   // UNICODE_TO_GBK[29826] := 16#8574;
   // UNICODE_TO_GBK[29827] := 16#D4CC;
   // UNICODE_TO_GBK[29828] := 16#8575;
   // UNICODE_TO_GBK[29829] := 16#CA98;
   // UNICODE_TO_GBK[29830] := 16#8576;
   // UNICODE_TO_GBK[29831] := 16#CA99;
   // UNICODE_TO_GBK[29832] := 16#8577;
   // UNICODE_TO_GBK[29833] := 16#CA9A;
   // UNICODE_TO_GBK[29834] := 16#8578;
   // UNICODE_TO_GBK[29835] := 16#CA9B;
   // UNICODE_TO_GBK[29836] := 16#8579;
   // UNICODE_TO_GBK[29837] := 16#DEB3;
   // UNICODE_TO_GBK[29838] := 16#857A;
   // UNICODE_TO_GBK[29839] := 16#DEAA;
   // UNICODE_TO_GBK[29840] := 16#857B;
   // UNICODE_TO_GBK[29841] := 16#DEAE;
   // UNICODE_TO_GBK[29842] := 16#857C;
   // UNICODE_TO_GBK[29843] := 16#CA9C;
   // UNICODE_TO_GBK[29844] := 16#857D;
   // UNICODE_TO_GBK[29845] := 16#CA9D;
   // UNICODE_TO_GBK[29846] := 16#857E;
   // UNICODE_TO_GBK[29847] := 16#C0D9;
   // UNICODE_TO_GBK[29848] := 16#857F;
   // UNICODE_TO_GBK[29849] := 16#CA9E;
   // UNICODE_TO_GBK[29850] := 16#8580;
   // UNICODE_TO_GBK[29851] := 16#CA9F;
   // UNICODE_TO_GBK[29852] := 16#8581;
   // UNICODE_TO_GBK[29853] := 16#CAA0;
   // UNICODE_TO_GBK[29854] := 16#8582;
   // UNICODE_TO_GBK[29855] := 16#CB40;
   // UNICODE_TO_GBK[29856] := 16#8583;
   // UNICODE_TO_GBK[29857] := 16#CB41;
   // UNICODE_TO_GBK[29858] := 16#8584;
   // UNICODE_TO_GBK[29859] := 16#B1A1;
   // UNICODE_TO_GBK[29860] := 16#8585;
   // UNICODE_TO_GBK[29861] := 16#DEB6;
   // UNICODE_TO_GBK[29862] := 16#8586;
   // UNICODE_TO_GBK[29863] := 16#CB42;
   // UNICODE_TO_GBK[29864] := 16#8587;
   // UNICODE_TO_GBK[29865] := 16#DEB1;
   // UNICODE_TO_GBK[29866] := 16#8588;
   // UNICODE_TO_GBK[29867] := 16#CB43;
   // UNICODE_TO_GBK[29868] := 16#8589;
   // UNICODE_TO_GBK[29869] := 16#CB44;
   // UNICODE_TO_GBK[29870] := 16#858A;
   // UNICODE_TO_GBK[29871] := 16#CB45;
   // UNICODE_TO_GBK[29872] := 16#858B;
   // UNICODE_TO_GBK[29873] := 16#CB46;
   // UNICODE_TO_GBK[29874] := 16#858C;
   // UNICODE_TO_GBK[29875] := 16#CB47;
   // UNICODE_TO_GBK[29876] := 16#858D;
   // UNICODE_TO_GBK[29877] := 16#CB48;
   // UNICODE_TO_GBK[29878] := 16#858E;
   // UNICODE_TO_GBK[29879] := 16#CB49;
   // UNICODE_TO_GBK[29880] := 16#858F;
   // UNICODE_TO_GBK[29881] := 16#DEB2;
   // UNICODE_TO_GBK[29882] := 16#8590;
   // UNICODE_TO_GBK[29883] := 16#CB4A;
   // UNICODE_TO_GBK[29884] := 16#8591;
   // UNICODE_TO_GBK[29885] := 16#CB4B;
   // UNICODE_TO_GBK[29886] := 16#8592;
   // UNICODE_TO_GBK[29887] := 16#CB4C;
   // UNICODE_TO_GBK[29888] := 16#8593;
   // UNICODE_TO_GBK[29889] := 16#CB4D;
   // UNICODE_TO_GBK[29890] := 16#8594;
   // UNICODE_TO_GBK[29891] := 16#CB4E;
   // UNICODE_TO_GBK[29892] := 16#8595;
   // UNICODE_TO_GBK[29893] := 16#CB4F;
   // UNICODE_TO_GBK[29894] := 16#8596;
   // UNICODE_TO_GBK[29895] := 16#CB50;
   // UNICODE_TO_GBK[29896] := 16#8597;
   // UNICODE_TO_GBK[29897] := 16#CB51;
   // UNICODE_TO_GBK[29898] := 16#8598;
   // UNICODE_TO_GBK[29899] := 16#CB52;
   // UNICODE_TO_GBK[29900] := 16#8599;
   // UNICODE_TO_GBK[29901] := 16#CB53;
   // UNICODE_TO_GBK[29902] := 16#859A;
   // UNICODE_TO_GBK[29903] := 16#CB54;
   // UNICODE_TO_GBK[29904] := 16#859B;
   // UNICODE_TO_GBK[29905] := 16#D1A6;
   // UNICODE_TO_GBK[29906] := 16#859C;
   // UNICODE_TO_GBK[29907] := 16#DEB5;
   // UNICODE_TO_GBK[29908] := 16#859D;
   // UNICODE_TO_GBK[29909] := 16#CB55;
   // UNICODE_TO_GBK[29910] := 16#859E;
   // UNICODE_TO_GBK[29911] := 16#CB56;
   // UNICODE_TO_GBK[29912] := 16#859F;
   // UNICODE_TO_GBK[29913] := 16#CB57;
   // UNICODE_TO_GBK[29914] := 16#85A0;
   // UNICODE_TO_GBK[29915] := 16#CB58;
   // UNICODE_TO_GBK[29916] := 16#85A1;
   // UNICODE_TO_GBK[29917] := 16#CB59;
   // UNICODE_TO_GBK[29918] := 16#85A2;
   // UNICODE_TO_GBK[29919] := 16#CB5A;
   // UNICODE_TO_GBK[29920] := 16#85A3;
   // UNICODE_TO_GBK[29921] := 16#CB5B;
   // UNICODE_TO_GBK[29922] := 16#85A4;
   // UNICODE_TO_GBK[29923] := 16#DEAF;
   // UNICODE_TO_GBK[29924] := 16#85A5;
   // UNICODE_TO_GBK[29925] := 16#CB5C;
   // UNICODE_TO_GBK[29926] := 16#85A6;
   // UNICODE_TO_GBK[29927] := 16#CB5D;
   // UNICODE_TO_GBK[29928] := 16#85A7;
   // UNICODE_TO_GBK[29929] := 16#CB5E;
   // UNICODE_TO_GBK[29930] := 16#85A8;
   // UNICODE_TO_GBK[29931] := 16#DEB0;
   // UNICODE_TO_GBK[29932] := 16#85A9;
   // UNICODE_TO_GBK[29933] := 16#CB5F;
   // UNICODE_TO_GBK[29934] := 16#85AA;
   // UNICODE_TO_GBK[29935] := 16#D0BD;
   // UNICODE_TO_GBK[29936] := 16#85AB;
   // UNICODE_TO_GBK[29937] := 16#CB60;
   // UNICODE_TO_GBK[29938] := 16#85AC;
   // UNICODE_TO_GBK[29939] := 16#CB61;
   // UNICODE_TO_GBK[29940] := 16#85AD;
   // UNICODE_TO_GBK[29941] := 16#CB62;
   // UNICODE_TO_GBK[29942] := 16#85AE;
   // UNICODE_TO_GBK[29943] := 16#DEB4;
   // UNICODE_TO_GBK[29944] := 16#85AF;
   // UNICODE_TO_GBK[29945] := 16#CAED;
   // UNICODE_TO_GBK[29946] := 16#85B0;
   // UNICODE_TO_GBK[29947] := 16#DEB9;
   // UNICODE_TO_GBK[29948] := 16#85B1;
   // UNICODE_TO_GBK[29949] := 16#CB63;
   // UNICODE_TO_GBK[29950] := 16#85B2;
   // UNICODE_TO_GBK[29951] := 16#CB64;
   // UNICODE_TO_GBK[29952] := 16#85B3;
   // UNICODE_TO_GBK[29953] := 16#CB65;
   // UNICODE_TO_GBK[29954] := 16#85B4;
   // UNICODE_TO_GBK[29955] := 16#CB66;
   // UNICODE_TO_GBK[29956] := 16#85B5;
   // UNICODE_TO_GBK[29957] := 16#CB67;
   // UNICODE_TO_GBK[29958] := 16#85B6;
   // UNICODE_TO_GBK[29959] := 16#CB68;
   // UNICODE_TO_GBK[29960] := 16#85B7;
   // UNICODE_TO_GBK[29961] := 16#DEB8;
   // UNICODE_TO_GBK[29962] := 16#85B8;
   // UNICODE_TO_GBK[29963] := 16#CB69;
   // UNICODE_TO_GBK[29964] := 16#85B9;
   // UNICODE_TO_GBK[29965] := 16#DEB7;
   // UNICODE_TO_GBK[29966] := 16#85BA;
   // UNICODE_TO_GBK[29967] := 16#CB6A;
   // UNICODE_TO_GBK[29968] := 16#85BB;
   // UNICODE_TO_GBK[29969] := 16#CB6B;
   // UNICODE_TO_GBK[29970] := 16#85BC;
   // UNICODE_TO_GBK[29971] := 16#CB6C;
   // UNICODE_TO_GBK[29972] := 16#85BD;
   // UNICODE_TO_GBK[29973] := 16#CB6D;
   // UNICODE_TO_GBK[29974] := 16#85BE;
   // UNICODE_TO_GBK[29975] := 16#CB6E;
   // UNICODE_TO_GBK[29976] := 16#85BF;
   // UNICODE_TO_GBK[29977] := 16#CB6F;
   // UNICODE_TO_GBK[29978] := 16#85C0;
   // UNICODE_TO_GBK[29979] := 16#CB70;
   // UNICODE_TO_GBK[29980] := 16#85C1;
   // UNICODE_TO_GBK[29981] := 16#DEBB;
   // UNICODE_TO_GBK[29982] := 16#85C2;
   // UNICODE_TO_GBK[29983] := 16#CB71;
   // UNICODE_TO_GBK[29984] := 16#85C3;
   // UNICODE_TO_GBK[29985] := 16#CB72;
   // UNICODE_TO_GBK[29986] := 16#85C4;
   // UNICODE_TO_GBK[29987] := 16#CB73;
   // UNICODE_TO_GBK[29988] := 16#85C5;
   // UNICODE_TO_GBK[29989] := 16#CB74;
   // UNICODE_TO_GBK[29990] := 16#85C6;
   // UNICODE_TO_GBK[29991] := 16#CB75;
   // UNICODE_TO_GBK[29992] := 16#85C7;
   // UNICODE_TO_GBK[29993] := 16#CB76;
   // UNICODE_TO_GBK[29994] := 16#85C8;
   // UNICODE_TO_GBK[29995] := 16#CB77;
   // UNICODE_TO_GBK[29996] := 16#85C9;
   // UNICODE_TO_GBK[29997] := 16#BDE5;
   // UNICODE_TO_GBK[29998] := 16#85CA;
   // UNICODE_TO_GBK[29999] := 16#CB78;
   // UNICODE_TO_GBK[30000] := 16#85CB;
   // UNICODE_TO_GBK[30001] := 16#CB79;
   // UNICODE_TO_GBK[30002] := 16#85CC;
   // UNICODE_TO_GBK[30003] := 16#CB7A;
   // UNICODE_TO_GBK[30004] := 16#85CD;
   // UNICODE_TO_GBK[30005] := 16#CB7B;
   // UNICODE_TO_GBK[30006] := 16#85CE;
   // UNICODE_TO_GBK[30007] := 16#CB7C;
   // UNICODE_TO_GBK[30008] := 16#85CF;
   // UNICODE_TO_GBK[30009] := 16#B2D8;
   // UNICODE_TO_GBK[30010] := 16#85D0;
   // UNICODE_TO_GBK[30011] := 16#C3EA;
   // UNICODE_TO_GBK[30012] := 16#85D1;
   // UNICODE_TO_GBK[30013] := 16#CB7D;
   // UNICODE_TO_GBK[30014] := 16#85D2;
   // UNICODE_TO_GBK[30015] := 16#CB7E;
   // UNICODE_TO_GBK[30016] := 16#85D3;
   // UNICODE_TO_GBK[30017] := 16#DEBA;
   // UNICODE_TO_GBK[30018] := 16#85D4;
   // UNICODE_TO_GBK[30019] := 16#CB80;
   // UNICODE_TO_GBK[30020] := 16#85D5;
   // UNICODE_TO_GBK[30021] := 16#C5BA;
   // UNICODE_TO_GBK[30022] := 16#85D6;
   // UNICODE_TO_GBK[30023] := 16#CB81;
   // UNICODE_TO_GBK[30024] := 16#85D7;
   // UNICODE_TO_GBK[30025] := 16#CB82;
   // UNICODE_TO_GBK[30026] := 16#85D8;
   // UNICODE_TO_GBK[30027] := 16#CB83;
   // UNICODE_TO_GBK[30028] := 16#85D9;
   // UNICODE_TO_GBK[30029] := 16#CB84;
   // UNICODE_TO_GBK[30030] := 16#85DA;
   // UNICODE_TO_GBK[30031] := 16#CB85;
   // UNICODE_TO_GBK[30032] := 16#85DB;
   // UNICODE_TO_GBK[30033] := 16#CB86;
   // UNICODE_TO_GBK[30034] := 16#85DC;
   // UNICODE_TO_GBK[30035] := 16#DEBC;
   // UNICODE_TO_GBK[30036] := 16#85DD;
   // UNICODE_TO_GBK[30037] := 16#CB87;
   // UNICODE_TO_GBK[30038] := 16#85DE;
   // UNICODE_TO_GBK[30039] := 16#CB88;
   // UNICODE_TO_GBK[30040] := 16#85DF;
   // UNICODE_TO_GBK[30041] := 16#CB89;
   // UNICODE_TO_GBK[30042] := 16#85E0;
   // UNICODE_TO_GBK[30043] := 16#CB8A;
   // UNICODE_TO_GBK[30044] := 16#85E1;
   // UNICODE_TO_GBK[30045] := 16#CB8B;
   // UNICODE_TO_GBK[30046] := 16#85E2;
   // UNICODE_TO_GBK[30047] := 16#CB8C;
   // UNICODE_TO_GBK[30048] := 16#85E3;
   // UNICODE_TO_GBK[30049] := 16#CB8D;
   // UNICODE_TO_GBK[30050] := 16#85E4;
   // UNICODE_TO_GBK[30051] := 16#CCD9;
   // UNICODE_TO_GBK[30052] := 16#85E5;
   // UNICODE_TO_GBK[30053] := 16#CB8E;
   // UNICODE_TO_GBK[30054] := 16#85E6;
   // UNICODE_TO_GBK[30055] := 16#CB8F;
   // UNICODE_TO_GBK[30056] := 16#85E7;
   // UNICODE_TO_GBK[30057] := 16#CB90;
   // UNICODE_TO_GBK[30058] := 16#85E8;
   // UNICODE_TO_GBK[30059] := 16#CB91;
   // UNICODE_TO_GBK[30060] := 16#85E9;
   // UNICODE_TO_GBK[30061] := 16#B7AA;
   // UNICODE_TO_GBK[30062] := 16#85EA;
   // UNICODE_TO_GBK[30063] := 16#CB92;
   // UNICODE_TO_GBK[30064] := 16#85EB;
   // UNICODE_TO_GBK[30065] := 16#CB93;
   // UNICODE_TO_GBK[30066] := 16#85EC;
   // UNICODE_TO_GBK[30067] := 16#CB94;
   // UNICODE_TO_GBK[30068] := 16#85ED;
   // UNICODE_TO_GBK[30069] := 16#CB95;
   // UNICODE_TO_GBK[30070] := 16#85EE;
   // UNICODE_TO_GBK[30071] := 16#CB96;
   // UNICODE_TO_GBK[30072] := 16#85EF;
   // UNICODE_TO_GBK[30073] := 16#CB97;
   // UNICODE_TO_GBK[30074] := 16#85F0;
   // UNICODE_TO_GBK[30075] := 16#CB98;
   // UNICODE_TO_GBK[30076] := 16#85F1;
   // UNICODE_TO_GBK[30077] := 16#CB99;
   // UNICODE_TO_GBK[30078] := 16#85F2;
   // UNICODE_TO_GBK[30079] := 16#CB9A;
   // UNICODE_TO_GBK[30080] := 16#85F3;
   // UNICODE_TO_GBK[30081] := 16#CB9B;
   // UNICODE_TO_GBK[30082] := 16#85F4;
   // UNICODE_TO_GBK[30083] := 16#CB9C;
   // UNICODE_TO_GBK[30084] := 16#85F5;
   // UNICODE_TO_GBK[30085] := 16#CB9D;
   // UNICODE_TO_GBK[30086] := 16#85F6;
   // UNICODE_TO_GBK[30087] := 16#CB9E;
   // UNICODE_TO_GBK[30088] := 16#85F7;
   // UNICODE_TO_GBK[30089] := 16#CB9F;
   // UNICODE_TO_GBK[30090] := 16#85F8;
   // UNICODE_TO_GBK[30091] := 16#CBA0;
   // UNICODE_TO_GBK[30092] := 16#85F9;
   // UNICODE_TO_GBK[30093] := 16#CC40;
   // UNICODE_TO_GBK[30094] := 16#85FA;
   // UNICODE_TO_GBK[30095] := 16#CC41;
   // UNICODE_TO_GBK[30096] := 16#85FB;
   // UNICODE_TO_GBK[30097] := 16#D4E5;
   // UNICODE_TO_GBK[30098] := 16#85FC;
   // UNICODE_TO_GBK[30099] := 16#CC42;
   // UNICODE_TO_GBK[30100] := 16#85FD;
   // UNICODE_TO_GBK[30101] := 16#CC43;
   // UNICODE_TO_GBK[30102] := 16#85FE;
   // UNICODE_TO_GBK[30103] := 16#CC44;
   // UNICODE_TO_GBK[30104] := 16#85FF;
   // UNICODE_TO_GBK[30105] := 16#DEBD;
   // UNICODE_TO_GBK[30106] := 16#8600;
   // UNICODE_TO_GBK[30107] := 16#CC45;
   // UNICODE_TO_GBK[30108] := 16#8601;
   // UNICODE_TO_GBK[30109] := 16#CC46;
   // UNICODE_TO_GBK[30110] := 16#8602;
   // UNICODE_TO_GBK[30111] := 16#CC47;
   // UNICODE_TO_GBK[30112] := 16#8603;
   // UNICODE_TO_GBK[30113] := 16#CC48;
   // UNICODE_TO_GBK[30114] := 16#8604;
   // UNICODE_TO_GBK[30115] := 16#CC49;
   // UNICODE_TO_GBK[30116] := 16#8605;
   // UNICODE_TO_GBK[30117] := 16#DEBF;
   // UNICODE_TO_GBK[30118] := 16#8606;
   // UNICODE_TO_GBK[30119] := 16#CC4A;
   // UNICODE_TO_GBK[30120] := 16#8607;
   // UNICODE_TO_GBK[30121] := 16#CC4B;
   // UNICODE_TO_GBK[30122] := 16#8608;
   // UNICODE_TO_GBK[30123] := 16#CC4C;
   // UNICODE_TO_GBK[30124] := 16#8609;
   // UNICODE_TO_GBK[30125] := 16#CC4D;
   // UNICODE_TO_GBK[30126] := 16#860A;
   // UNICODE_TO_GBK[30127] := 16#CC4E;
   // UNICODE_TO_GBK[30128] := 16#860B;
   // UNICODE_TO_GBK[30129] := 16#CC4F;
   // UNICODE_TO_GBK[30130] := 16#860C;
   // UNICODE_TO_GBK[30131] := 16#CC50;
   // UNICODE_TO_GBK[30132] := 16#860D;
   // UNICODE_TO_GBK[30133] := 16#CC51;
   // UNICODE_TO_GBK[30134] := 16#860E;
   // UNICODE_TO_GBK[30135] := 16#CC52;
   // UNICODE_TO_GBK[30136] := 16#860F;
   // UNICODE_TO_GBK[30137] := 16#CC53;
   // UNICODE_TO_GBK[30138] := 16#8610;
   // UNICODE_TO_GBK[30139] := 16#CC54;
   // UNICODE_TO_GBK[30140] := 16#8611;
   // UNICODE_TO_GBK[30141] := 16#C4A2;
   // UNICODE_TO_GBK[30142] := 16#8612;
   // UNICODE_TO_GBK[30143] := 16#CC55;
   // UNICODE_TO_GBK[30144] := 16#8613;
   // UNICODE_TO_GBK[30145] := 16#CC56;
   // UNICODE_TO_GBK[30146] := 16#8614;
   // UNICODE_TO_GBK[30147] := 16#CC57;
   // UNICODE_TO_GBK[30148] := 16#8615;
   // UNICODE_TO_GBK[30149] := 16#CC58;
   // UNICODE_TO_GBK[30150] := 16#8616;
   // UNICODE_TO_GBK[30151] := 16#DEC1;
   // UNICODE_TO_GBK[30152] := 16#8617;
   // UNICODE_TO_GBK[30153] := 16#CC59;
   // UNICODE_TO_GBK[30154] := 16#8618;
   // UNICODE_TO_GBK[30155] := 16#CC5A;
   // UNICODE_TO_GBK[30156] := 16#8619;
   // UNICODE_TO_GBK[30157] := 16#CC5B;
   // UNICODE_TO_GBK[30158] := 16#861A;
   // UNICODE_TO_GBK[30159] := 16#CC5C;
   // UNICODE_TO_GBK[30160] := 16#861B;
   // UNICODE_TO_GBK[30161] := 16#CC5D;
   // UNICODE_TO_GBK[30162] := 16#861C;
   // UNICODE_TO_GBK[30163] := 16#CC5E;
   // UNICODE_TO_GBK[30164] := 16#861D;
   // UNICODE_TO_GBK[30165] := 16#CC5F;
   // UNICODE_TO_GBK[30166] := 16#861E;
   // UNICODE_TO_GBK[30167] := 16#CC60;
   // UNICODE_TO_GBK[30168] := 16#861F;
   // UNICODE_TO_GBK[30169] := 16#CC61;
   // UNICODE_TO_GBK[30170] := 16#8620;
   // UNICODE_TO_GBK[30171] := 16#CC62;
   // UNICODE_TO_GBK[30172] := 16#8621;
   // UNICODE_TO_GBK[30173] := 16#CC63;
   // UNICODE_TO_GBK[30174] := 16#8622;
   // UNICODE_TO_GBK[30175] := 16#CC64;
   // UNICODE_TO_GBK[30176] := 16#8623;
   // UNICODE_TO_GBK[30177] := 16#CC65;
   // UNICODE_TO_GBK[30178] := 16#8624;
   // UNICODE_TO_GBK[30179] := 16#CC66;
   // UNICODE_TO_GBK[30180] := 16#8625;
   // UNICODE_TO_GBK[30181] := 16#CC67;
   // UNICODE_TO_GBK[30182] := 16#8626;
   // UNICODE_TO_GBK[30183] := 16#CC68;
   // UNICODE_TO_GBK[30184] := 16#8627;
   // UNICODE_TO_GBK[30185] := 16#DEBE;
   // UNICODE_TO_GBK[30186] := 16#8628;
   // UNICODE_TO_GBK[30187] := 16#CC69;
   // UNICODE_TO_GBK[30188] := 16#8629;
   // UNICODE_TO_GBK[30189] := 16#DEC0;
   // UNICODE_TO_GBK[30190] := 16#862A;
   // UNICODE_TO_GBK[30191] := 16#CC6A;
   // UNICODE_TO_GBK[30192] := 16#862B;
   // UNICODE_TO_GBK[30193] := 16#CC6B;
   // UNICODE_TO_GBK[30194] := 16#862C;
   // UNICODE_TO_GBK[30195] := 16#CC6C;
   // UNICODE_TO_GBK[30196] := 16#862D;
   // UNICODE_TO_GBK[30197] := 16#CC6D;
   // UNICODE_TO_GBK[30198] := 16#862E;
   // UNICODE_TO_GBK[30199] := 16#CC6E;
   // UNICODE_TO_GBK[30200] := 16#862F;
   // UNICODE_TO_GBK[30201] := 16#CC6F;
   // UNICODE_TO_GBK[30202] := 16#8630;
   // UNICODE_TO_GBK[30203] := 16#CC70;
   // UNICODE_TO_GBK[30204] := 16#8631;
   // UNICODE_TO_GBK[30205] := 16#CC71;
   // UNICODE_TO_GBK[30206] := 16#8632;
   // UNICODE_TO_GBK[30207] := 16#CC72;
   // UNICODE_TO_GBK[30208] := 16#8633;
   // UNICODE_TO_GBK[30209] := 16#CC73;
   // UNICODE_TO_GBK[30210] := 16#8634;
   // UNICODE_TO_GBK[30211] := 16#CC74;
   // UNICODE_TO_GBK[30212] := 16#8635;
   // UNICODE_TO_GBK[30213] := 16#CC75;
   // UNICODE_TO_GBK[30214] := 16#8636;
   // UNICODE_TO_GBK[30215] := 16#CC76;
   // UNICODE_TO_GBK[30216] := 16#8637;
   // UNICODE_TO_GBK[30217] := 16#CC77;
   // UNICODE_TO_GBK[30218] := 16#8638;
   // UNICODE_TO_GBK[30219] := 16#D5BA;
   // UNICODE_TO_GBK[30220] := 16#8639;
   // UNICODE_TO_GBK[30221] := 16#CC78;
   // UNICODE_TO_GBK[30222] := 16#863A;
   // UNICODE_TO_GBK[30223] := 16#CC79;
   // UNICODE_TO_GBK[30224] := 16#863B;
   // UNICODE_TO_GBK[30225] := 16#CC7A;
   // UNICODE_TO_GBK[30226] := 16#863C;
   // UNICODE_TO_GBK[30227] := 16#DEC2;
   // UNICODE_TO_GBK[30228] := 16#863D;
   // UNICODE_TO_GBK[30229] := 16#CC7B;
   // UNICODE_TO_GBK[30230] := 16#863E;
   // UNICODE_TO_GBK[30231] := 16#CC7C;
   // UNICODE_TO_GBK[30232] := 16#863F;
   // UNICODE_TO_GBK[30233] := 16#CC7D;
   // UNICODE_TO_GBK[30234] := 16#8640;
   // UNICODE_TO_GBK[30235] := 16#CC7E;
   // UNICODE_TO_GBK[30236] := 16#8641;
   // UNICODE_TO_GBK[30237] := 16#CC80;
   // UNICODE_TO_GBK[30238] := 16#8642;
   // UNICODE_TO_GBK[30239] := 16#CC81;
   // UNICODE_TO_GBK[30240] := 16#8643;
   // UNICODE_TO_GBK[30241] := 16#CC82;
   // UNICODE_TO_GBK[30242] := 16#8644;
   // UNICODE_TO_GBK[30243] := 16#CC83;
   // UNICODE_TO_GBK[30244] := 16#8645;
   // UNICODE_TO_GBK[30245] := 16#CC84;
   // UNICODE_TO_GBK[30246] := 16#8646;
   // UNICODE_TO_GBK[30247] := 16#CC85;
   // UNICODE_TO_GBK[30248] := 16#8647;
   // UNICODE_TO_GBK[30249] := 16#CC86;
   // UNICODE_TO_GBK[30250] := 16#8648;
   // UNICODE_TO_GBK[30251] := 16#CC87;
   // UNICODE_TO_GBK[30252] := 16#8649;
   // UNICODE_TO_GBK[30253] := 16#CC88;
   // UNICODE_TO_GBK[30254] := 16#864A;
   // UNICODE_TO_GBK[30255] := 16#CC89;
   // UNICODE_TO_GBK[30256] := 16#864B;
   // UNICODE_TO_GBK[30257] := 16#CC8A;
   // UNICODE_TO_GBK[30258] := 16#864C;
   // UNICODE_TO_GBK[30259] := 16#CC8B;
   // UNICODE_TO_GBK[30260] := 16#864D;
   // UNICODE_TO_GBK[30261] := 16#F2AE;
   // UNICODE_TO_GBK[30262] := 16#864E;
   // UNICODE_TO_GBK[30263] := 16#BBA2;
   // UNICODE_TO_GBK[30264] := 16#864F;
   // UNICODE_TO_GBK[30265] := 16#C2B2;
   // UNICODE_TO_GBK[30266] := 16#8650;
   // UNICODE_TO_GBK[30267] := 16#C5B0;
   // UNICODE_TO_GBK[30268] := 16#8651;
   // UNICODE_TO_GBK[30269] := 16#C2C7;
   // UNICODE_TO_GBK[30270] := 16#8652;
   // UNICODE_TO_GBK[30271] := 16#CC8C;
   // UNICODE_TO_GBK[30272] := 16#8653;
   // UNICODE_TO_GBK[30273] := 16#CC8D;
   // UNICODE_TO_GBK[30274] := 16#8654;
   // UNICODE_TO_GBK[30275] := 16#F2AF;
   // UNICODE_TO_GBK[30276] := 16#8655;
   // UNICODE_TO_GBK[30277] := 16#CC8E;
   // UNICODE_TO_GBK[30278] := 16#8656;
   // UNICODE_TO_GBK[30279] := 16#CC8F;
   // UNICODE_TO_GBK[30280] := 16#8657;
   // UNICODE_TO_GBK[30281] := 16#CC90;
   // UNICODE_TO_GBK[30282] := 16#8658;
   // UNICODE_TO_GBK[30283] := 16#CC91;
   // UNICODE_TO_GBK[30284] := 16#8659;
   // UNICODE_TO_GBK[30285] := 16#CC92;
   // UNICODE_TO_GBK[30286] := 16#865A;
   // UNICODE_TO_GBK[30287] := 16#D0E9;
   // UNICODE_TO_GBK[30288] := 16#865B;
   // UNICODE_TO_GBK[30289] := 16#CC93;
   // UNICODE_TO_GBK[30290] := 16#865C;
   // UNICODE_TO_GBK[30291] := 16#CC94;
   // UNICODE_TO_GBK[30292] := 16#865D;
   // UNICODE_TO_GBK[30293] := 16#CC95;
   // UNICODE_TO_GBK[30294] := 16#865E;
   // UNICODE_TO_GBK[30295] := 16#D3DD;
   // UNICODE_TO_GBK[30296] := 16#865F;
   // UNICODE_TO_GBK[30297] := 16#CC96;
   // UNICODE_TO_GBK[30298] := 16#8660;
   // UNICODE_TO_GBK[30299] := 16#CC97;
   // UNICODE_TO_GBK[30300] := 16#8661;
   // UNICODE_TO_GBK[30301] := 16#CC98;
   // UNICODE_TO_GBK[30302] := 16#8662;
   // UNICODE_TO_GBK[30303] := 16#EBBD;
   // UNICODE_TO_GBK[30304] := 16#8663;
   // UNICODE_TO_GBK[30305] := 16#CC99;
   // UNICODE_TO_GBK[30306] := 16#8664;
   // UNICODE_TO_GBK[30307] := 16#CC9A;
   // UNICODE_TO_GBK[30308] := 16#8665;
   // UNICODE_TO_GBK[30309] := 16#CC9B;
   // UNICODE_TO_GBK[30310] := 16#8666;
   // UNICODE_TO_GBK[30311] := 16#CC9C;
   // UNICODE_TO_GBK[30312] := 16#8667;
   // UNICODE_TO_GBK[30313] := 16#CC9D;
   // UNICODE_TO_GBK[30314] := 16#8668;
   // UNICODE_TO_GBK[30315] := 16#CC9E;
   // UNICODE_TO_GBK[30316] := 16#8669;
   // UNICODE_TO_GBK[30317] := 16#CC9F;
   // UNICODE_TO_GBK[30318] := 16#866A;
   // UNICODE_TO_GBK[30319] := 16#CCA0;
   // UNICODE_TO_GBK[30320] := 16#866B;
   // UNICODE_TO_GBK[30321] := 16#B3E6;
   // UNICODE_TO_GBK[30322] := 16#866C;
   // UNICODE_TO_GBK[30323] := 16#F2B0;
   // UNICODE_TO_GBK[30324] := 16#866D;
   // UNICODE_TO_GBK[30325] := 16#CD40;
   // UNICODE_TO_GBK[30326] := 16#866E;
   // UNICODE_TO_GBK[30327] := 16#F2B1;
   // UNICODE_TO_GBK[30328] := 16#866F;
   // UNICODE_TO_GBK[30329] := 16#CD41;
   // UNICODE_TO_GBK[30330] := 16#8670;
   // UNICODE_TO_GBK[30331] := 16#CD42;
   // UNICODE_TO_GBK[30332] := 16#8671;
   // UNICODE_TO_GBK[30333] := 16#CAAD;
   // UNICODE_TO_GBK[30334] := 16#8672;
   // UNICODE_TO_GBK[30335] := 16#CD43;
   // UNICODE_TO_GBK[30336] := 16#8673;
   // UNICODE_TO_GBK[30337] := 16#CD44;
   // UNICODE_TO_GBK[30338] := 16#8674;
   // UNICODE_TO_GBK[30339] := 16#CD45;
   // UNICODE_TO_GBK[30340] := 16#8675;
   // UNICODE_TO_GBK[30341] := 16#CD46;
   // UNICODE_TO_GBK[30342] := 16#8676;
   // UNICODE_TO_GBK[30343] := 16#CD47;
   // UNICODE_TO_GBK[30344] := 16#8677;
   // UNICODE_TO_GBK[30345] := 16#CD48;
   // UNICODE_TO_GBK[30346] := 16#8678;
   // UNICODE_TO_GBK[30347] := 16#CD49;
   // UNICODE_TO_GBK[30348] := 16#8679;
   // UNICODE_TO_GBK[30349] := 16#BAE7;
   // UNICODE_TO_GBK[30350] := 16#867A;
   // UNICODE_TO_GBK[30351] := 16#F2B3;
   // UNICODE_TO_GBK[30352] := 16#867B;
   // UNICODE_TO_GBK[30353] := 16#F2B5;
   // UNICODE_TO_GBK[30354] := 16#867C;
   // UNICODE_TO_GBK[30355] := 16#F2B4;
   // UNICODE_TO_GBK[30356] := 16#867D;
   // UNICODE_TO_GBK[30357] := 16#CBE4;
   // UNICODE_TO_GBK[30358] := 16#867E;
   // UNICODE_TO_GBK[30359] := 16#CFBA;
   // UNICODE_TO_GBK[30360] := 16#867F;
   // UNICODE_TO_GBK[30361] := 16#F2B2;
   // UNICODE_TO_GBK[30362] := 16#8680;
   // UNICODE_TO_GBK[30363] := 16#CAB4;
   // UNICODE_TO_GBK[30364] := 16#8681;
   // UNICODE_TO_GBK[30365] := 16#D2CF;
   // UNICODE_TO_GBK[30366] := 16#8682;
   // UNICODE_TO_GBK[30367] := 16#C2EC;
   // UNICODE_TO_GBK[30368] := 16#8683;
   // UNICODE_TO_GBK[30369] := 16#CD4A;
   // UNICODE_TO_GBK[30370] := 16#8684;
   // UNICODE_TO_GBK[30371] := 16#CD4B;
   // UNICODE_TO_GBK[30372] := 16#8685;
   // UNICODE_TO_GBK[30373] := 16#CD4C;
   // UNICODE_TO_GBK[30374] := 16#8686;
   // UNICODE_TO_GBK[30375] := 16#CD4D;
   // UNICODE_TO_GBK[30376] := 16#8687;
   // UNICODE_TO_GBK[30377] := 16#CD4E;
   // UNICODE_TO_GBK[30378] := 16#8688;
   // UNICODE_TO_GBK[30379] := 16#CD4F;
   // UNICODE_TO_GBK[30380] := 16#8689;
   // UNICODE_TO_GBK[30381] := 16#CD50;
   // UNICODE_TO_GBK[30382] := 16#868A;
   // UNICODE_TO_GBK[30383] := 16#CEC3;
   // UNICODE_TO_GBK[30384] := 16#868B;
   // UNICODE_TO_GBK[30385] := 16#F2B8;
   // UNICODE_TO_GBK[30386] := 16#868C;
   // UNICODE_TO_GBK[30387] := 16#B0F6;
   // UNICODE_TO_GBK[30388] := 16#868D;
   // UNICODE_TO_GBK[30389] := 16#F2B7;
   // UNICODE_TO_GBK[30390] := 16#868E;
   // UNICODE_TO_GBK[30391] := 16#CD51;
   // UNICODE_TO_GBK[30392] := 16#868F;
   // UNICODE_TO_GBK[30393] := 16#CD52;
   // UNICODE_TO_GBK[30394] := 16#8690;
   // UNICODE_TO_GBK[30395] := 16#CD53;
   // UNICODE_TO_GBK[30396] := 16#8691;
   // UNICODE_TO_GBK[30397] := 16#CD54;
   // UNICODE_TO_GBK[30398] := 16#8692;
   // UNICODE_TO_GBK[30399] := 16#CD55;
   // UNICODE_TO_GBK[30400] := 16#8693;
   // UNICODE_TO_GBK[30401] := 16#F2BE;
   // UNICODE_TO_GBK[30402] := 16#8694;
   // UNICODE_TO_GBK[30403] := 16#CD56;
   // UNICODE_TO_GBK[30404] := 16#8695;
   // UNICODE_TO_GBK[30405] := 16#B2CF;
   // UNICODE_TO_GBK[30406] := 16#8696;
   // UNICODE_TO_GBK[30407] := 16#CD57;
   // UNICODE_TO_GBK[30408] := 16#8697;
   // UNICODE_TO_GBK[30409] := 16#CD58;
   // UNICODE_TO_GBK[30410] := 16#8698;
   // UNICODE_TO_GBK[30411] := 16#CD59;
   // UNICODE_TO_GBK[30412] := 16#8699;
   // UNICODE_TO_GBK[30413] := 16#CD5A;
   // UNICODE_TO_GBK[30414] := 16#869A;
   // UNICODE_TO_GBK[30415] := 16#CD5B;
   // UNICODE_TO_GBK[30416] := 16#869B;
   // UNICODE_TO_GBK[30417] := 16#CD5C;
   // UNICODE_TO_GBK[30418] := 16#869C;
   // UNICODE_TO_GBK[30419] := 16#D1C1;
   // UNICODE_TO_GBK[30420] := 16#869D;
   // UNICODE_TO_GBK[30421] := 16#F2BA;
   // UNICODE_TO_GBK[30422] := 16#869E;
   // UNICODE_TO_GBK[30423] := 16#CD5D;
   // UNICODE_TO_GBK[30424] := 16#869F;
   // UNICODE_TO_GBK[30425] := 16#CD5E;
   // UNICODE_TO_GBK[30426] := 16#86A0;
   // UNICODE_TO_GBK[30427] := 16#CD5F;
   // UNICODE_TO_GBK[30428] := 16#86A1;
   // UNICODE_TO_GBK[30429] := 16#CD60;
   // UNICODE_TO_GBK[30430] := 16#86A2;
   // UNICODE_TO_GBK[30431] := 16#CD61;
   // UNICODE_TO_GBK[30432] := 16#86A3;
   // UNICODE_TO_GBK[30433] := 16#F2BC;
   // UNICODE_TO_GBK[30434] := 16#86A4;
   // UNICODE_TO_GBK[30435] := 16#D4E9;
   // UNICODE_TO_GBK[30436] := 16#86A5;
   // UNICODE_TO_GBK[30437] := 16#CD62;
   // UNICODE_TO_GBK[30438] := 16#86A6;
   // UNICODE_TO_GBK[30439] := 16#CD63;
   // UNICODE_TO_GBK[30440] := 16#86A7;
   // UNICODE_TO_GBK[30441] := 16#F2BB;
   // UNICODE_TO_GBK[30442] := 16#86A8;
   // UNICODE_TO_GBK[30443] := 16#F2B6;
   // UNICODE_TO_GBK[30444] := 16#86A9;
   // UNICODE_TO_GBK[30445] := 16#F2BF;
   // UNICODE_TO_GBK[30446] := 16#86AA;
   // UNICODE_TO_GBK[30447] := 16#F2BD;
   // UNICODE_TO_GBK[30448] := 16#86AB;
   // UNICODE_TO_GBK[30449] := 16#CD64;
   // UNICODE_TO_GBK[30450] := 16#86AC;
   // UNICODE_TO_GBK[30451] := 16#F2B9;
   // UNICODE_TO_GBK[30452] := 16#86AD;
   // UNICODE_TO_GBK[30453] := 16#CD65;
   // UNICODE_TO_GBK[30454] := 16#86AE;
   // UNICODE_TO_GBK[30455] := 16#CD66;
   // UNICODE_TO_GBK[30456] := 16#86AF;
   // UNICODE_TO_GBK[30457] := 16#F2C7;
   // UNICODE_TO_GBK[30458] := 16#86B0;
   // UNICODE_TO_GBK[30459] := 16#F2C4;
   // UNICODE_TO_GBK[30460] := 16#86B1;
   // UNICODE_TO_GBK[30461] := 16#F2C6;
   // UNICODE_TO_GBK[30462] := 16#86B2;
   // UNICODE_TO_GBK[30463] := 16#CD67;
   // UNICODE_TO_GBK[30464] := 16#86B3;
   // UNICODE_TO_GBK[30465] := 16#CD68;
   // UNICODE_TO_GBK[30466] := 16#86B4;
   // UNICODE_TO_GBK[30467] := 16#F2CA;
   // UNICODE_TO_GBK[30468] := 16#86B5;
   // UNICODE_TO_GBK[30469] := 16#F2C2;
   // UNICODE_TO_GBK[30470] := 16#86B6;
   // UNICODE_TO_GBK[30471] := 16#F2C0;
   // UNICODE_TO_GBK[30472] := 16#86B7;
   // UNICODE_TO_GBK[30473] := 16#CD69;
   // UNICODE_TO_GBK[30474] := 16#86B8;
   // UNICODE_TO_GBK[30475] := 16#CD6A;
   // UNICODE_TO_GBK[30476] := 16#86B9;
   // UNICODE_TO_GBK[30477] := 16#CD6B;
   // UNICODE_TO_GBK[30478] := 16#86BA;
   // UNICODE_TO_GBK[30479] := 16#F2C5;
   // UNICODE_TO_GBK[30480] := 16#86BB;
   // UNICODE_TO_GBK[30481] := 16#CD6C;
   // UNICODE_TO_GBK[30482] := 16#86BC;
   // UNICODE_TO_GBK[30483] := 16#CD6D;
   // UNICODE_TO_GBK[30484] := 16#86BD;
   // UNICODE_TO_GBK[30485] := 16#CD6E;
   // UNICODE_TO_GBK[30486] := 16#86BE;
   // UNICODE_TO_GBK[30487] := 16#CD6F;
   // UNICODE_TO_GBK[30488] := 16#86BF;
   // UNICODE_TO_GBK[30489] := 16#CD70;
   // UNICODE_TO_GBK[30490] := 16#86C0;
   // UNICODE_TO_GBK[30491] := 16#D6FB;
   // UNICODE_TO_GBK[30492] := 16#86C1;
   // UNICODE_TO_GBK[30493] := 16#CD71;
   // UNICODE_TO_GBK[30494] := 16#86C2;
   // UNICODE_TO_GBK[30495] := 16#CD72;
   // UNICODE_TO_GBK[30496] := 16#86C3;
   // UNICODE_TO_GBK[30497] := 16#CD73;
   // UNICODE_TO_GBK[30498] := 16#86C4;
   // UNICODE_TO_GBK[30499] := 16#F2C1;
   // UNICODE_TO_GBK[30500] := 16#86C5;
   // UNICODE_TO_GBK[30501] := 16#CD74;
   // UNICODE_TO_GBK[30502] := 16#86C6;
   // UNICODE_TO_GBK[30503] := 16#C7F9;
   // UNICODE_TO_GBK[30504] := 16#86C7;
   // UNICODE_TO_GBK[30505] := 16#C9DF;
   // UNICODE_TO_GBK[30506] := 16#86C8;
   // UNICODE_TO_GBK[30507] := 16#CD75;
   // UNICODE_TO_GBK[30508] := 16#86C9;
   // UNICODE_TO_GBK[30509] := 16#F2C8;
   // UNICODE_TO_GBK[30510] := 16#86CA;
   // UNICODE_TO_GBK[30511] := 16#B9C6;
   // UNICODE_TO_GBK[30512] := 16#86CB;
   // UNICODE_TO_GBK[30513] := 16#B5B0;
   // UNICODE_TO_GBK[30514] := 16#86CC;
   // UNICODE_TO_GBK[30515] := 16#CD76;
   // UNICODE_TO_GBK[30516] := 16#86CD;
   // UNICODE_TO_GBK[30517] := 16#CD77;
   // UNICODE_TO_GBK[30518] := 16#86CE;
   // UNICODE_TO_GBK[30519] := 16#F2C3;
   // UNICODE_TO_GBK[30520] := 16#86CF;
   // UNICODE_TO_GBK[30521] := 16#F2C9;
   // UNICODE_TO_GBK[30522] := 16#86D0;
   // UNICODE_TO_GBK[30523] := 16#F2D0;
   // UNICODE_TO_GBK[30524] := 16#86D1;
   // UNICODE_TO_GBK[30525] := 16#F2D6;
   // UNICODE_TO_GBK[30526] := 16#86D2;
   // UNICODE_TO_GBK[30527] := 16#CD78;
   // UNICODE_TO_GBK[30528] := 16#86D3;
   // UNICODE_TO_GBK[30529] := 16#CD79;
   // UNICODE_TO_GBK[30530] := 16#86D4;
   // UNICODE_TO_GBK[30531] := 16#BBD7;
   // UNICODE_TO_GBK[30532] := 16#86D5;
   // UNICODE_TO_GBK[30533] := 16#CD7A;
   // UNICODE_TO_GBK[30534] := 16#86D6;
   // UNICODE_TO_GBK[30535] := 16#CD7B;
   // UNICODE_TO_GBK[30536] := 16#86D7;
   // UNICODE_TO_GBK[30537] := 16#CD7C;
   // UNICODE_TO_GBK[30538] := 16#86D8;
   // UNICODE_TO_GBK[30539] := 16#F2D5;
   // UNICODE_TO_GBK[30540] := 16#86D9;
   // UNICODE_TO_GBK[30541] := 16#CDDC;
   // UNICODE_TO_GBK[30542] := 16#86DA;
   // UNICODE_TO_GBK[30543] := 16#CD7D;
   // UNICODE_TO_GBK[30544] := 16#86DB;
   // UNICODE_TO_GBK[30545] := 16#D6EB;
   // UNICODE_TO_GBK[30546] := 16#86DC;
   // UNICODE_TO_GBK[30547] := 16#CD7E;
   // UNICODE_TO_GBK[30548] := 16#86DD;
   // UNICODE_TO_GBK[30549] := 16#CD80;
   // UNICODE_TO_GBK[30550] := 16#86DE;
   // UNICODE_TO_GBK[30551] := 16#F2D2;
   // UNICODE_TO_GBK[30552] := 16#86DF;
   // UNICODE_TO_GBK[30553] := 16#F2D4;
   // UNICODE_TO_GBK[30554] := 16#86E0;
   // UNICODE_TO_GBK[30555] := 16#CD81;
   // UNICODE_TO_GBK[30556] := 16#86E1;
   // UNICODE_TO_GBK[30557] := 16#CD82;
   // UNICODE_TO_GBK[30558] := 16#86E2;
   // UNICODE_TO_GBK[30559] := 16#CD83;
   // UNICODE_TO_GBK[30560] := 16#86E3;
   // UNICODE_TO_GBK[30561] := 16#CD84;
   // UNICODE_TO_GBK[30562] := 16#86E4;
   // UNICODE_TO_GBK[30563] := 16#B8F2;
   // UNICODE_TO_GBK[30564] := 16#86E5;
   // UNICODE_TO_GBK[30565] := 16#CD85;
   // UNICODE_TO_GBK[30566] := 16#86E6;
   // UNICODE_TO_GBK[30567] := 16#CD86;
   // UNICODE_TO_GBK[30568] := 16#86E7;
   // UNICODE_TO_GBK[30569] := 16#CD87;
   // UNICODE_TO_GBK[30570] := 16#86E8;
   // UNICODE_TO_GBK[30571] := 16#CD88;
   // UNICODE_TO_GBK[30572] := 16#86E9;
   // UNICODE_TO_GBK[30573] := 16#F2CB;
   // UNICODE_TO_GBK[30574] := 16#86EA;
   // UNICODE_TO_GBK[30575] := 16#CD89;
   // UNICODE_TO_GBK[30576] := 16#86EB;
   // UNICODE_TO_GBK[30577] := 16#CD8A;
   // UNICODE_TO_GBK[30578] := 16#86EC;
   // UNICODE_TO_GBK[30579] := 16#CD8B;
   // UNICODE_TO_GBK[30580] := 16#86ED;
   // UNICODE_TO_GBK[30581] := 16#F2CE;
   // UNICODE_TO_GBK[30582] := 16#86EE;
   // UNICODE_TO_GBK[30583] := 16#C2F9;
   // UNICODE_TO_GBK[30584] := 16#86EF;
   // UNICODE_TO_GBK[30585] := 16#CD8C;
   // UNICODE_TO_GBK[30586] := 16#86F0;
   // UNICODE_TO_GBK[30587] := 16#D5DD;
   // UNICODE_TO_GBK[30588] := 16#86F1;
   // UNICODE_TO_GBK[30589] := 16#F2CC;
   // UNICODE_TO_GBK[30590] := 16#86F2;
   // UNICODE_TO_GBK[30591] := 16#F2CD;
   // UNICODE_TO_GBK[30592] := 16#86F3;
   // UNICODE_TO_GBK[30593] := 16#F2CF;
   // UNICODE_TO_GBK[30594] := 16#86F4;
   // UNICODE_TO_GBK[30595] := 16#F2D3;
   // UNICODE_TO_GBK[30596] := 16#86F5;
   // UNICODE_TO_GBK[30597] := 16#CD8D;
   // UNICODE_TO_GBK[30598] := 16#86F6;
   // UNICODE_TO_GBK[30599] := 16#CD8E;
   // UNICODE_TO_GBK[30600] := 16#86F7;
   // UNICODE_TO_GBK[30601] := 16#CD8F;
   // UNICODE_TO_GBK[30602] := 16#86F8;
   // UNICODE_TO_GBK[30603] := 16#F2D9;
   // UNICODE_TO_GBK[30604] := 16#86F9;
   // UNICODE_TO_GBK[30605] := 16#D3BC;
   // UNICODE_TO_GBK[30606] := 16#86FA;
   // UNICODE_TO_GBK[30607] := 16#CD90;
   // UNICODE_TO_GBK[30608] := 16#86FB;
   // UNICODE_TO_GBK[30609] := 16#CD91;
   // UNICODE_TO_GBK[30610] := 16#86FC;
   // UNICODE_TO_GBK[30611] := 16#CD92;
   // UNICODE_TO_GBK[30612] := 16#86FD;
   // UNICODE_TO_GBK[30613] := 16#CD93;
   // UNICODE_TO_GBK[30614] := 16#86FE;
   // UNICODE_TO_GBK[30615] := 16#B6EA;
   // UNICODE_TO_GBK[30616] := 16#86FF;
   // UNICODE_TO_GBK[30617] := 16#CD94;
   // UNICODE_TO_GBK[30618] := 16#8700;
   // UNICODE_TO_GBK[30619] := 16#CAF1;
   // UNICODE_TO_GBK[30620] := 16#8701;
   // UNICODE_TO_GBK[30621] := 16#CD95;
   // UNICODE_TO_GBK[30622] := 16#8702;
   // UNICODE_TO_GBK[30623] := 16#B7E4;
   // UNICODE_TO_GBK[30624] := 16#8703;
   // UNICODE_TO_GBK[30625] := 16#F2D7;
   // UNICODE_TO_GBK[30626] := 16#8704;
   // UNICODE_TO_GBK[30627] := 16#CD96;
   // UNICODE_TO_GBK[30628] := 16#8705;
   // UNICODE_TO_GBK[30629] := 16#CD97;
   // UNICODE_TO_GBK[30630] := 16#8706;
   // UNICODE_TO_GBK[30631] := 16#CD98;
   // UNICODE_TO_GBK[30632] := 16#8707;
   // UNICODE_TO_GBK[30633] := 16#F2D8;
   // UNICODE_TO_GBK[30634] := 16#8708;
   // UNICODE_TO_GBK[30635] := 16#F2DA;
   // UNICODE_TO_GBK[30636] := 16#8709;
   // UNICODE_TO_GBK[30637] := 16#F2DD;
   // UNICODE_TO_GBK[30638] := 16#870A;
   // UNICODE_TO_GBK[30639] := 16#F2DB;
   // UNICODE_TO_GBK[30640] := 16#870B;
   // UNICODE_TO_GBK[30641] := 16#CD99;
   // UNICODE_TO_GBK[30642] := 16#870C;
   // UNICODE_TO_GBK[30643] := 16#CD9A;
   // UNICODE_TO_GBK[30644] := 16#870D;
   // UNICODE_TO_GBK[30645] := 16#F2DC;
   // UNICODE_TO_GBK[30646] := 16#870E;
   // UNICODE_TO_GBK[30647] := 16#CD9B;
   // UNICODE_TO_GBK[30648] := 16#870F;
   // UNICODE_TO_GBK[30649] := 16#CD9C;
   // UNICODE_TO_GBK[30650] := 16#8710;
   // UNICODE_TO_GBK[30651] := 16#CD9D;
   // UNICODE_TO_GBK[30652] := 16#8711;
   // UNICODE_TO_GBK[30653] := 16#CD9E;
   // UNICODE_TO_GBK[30654] := 16#8712;
   // UNICODE_TO_GBK[30655] := 16#D1D1;
   // UNICODE_TO_GBK[30656] := 16#8713;
   // UNICODE_TO_GBK[30657] := 16#F2D1;
   // UNICODE_TO_GBK[30658] := 16#8714;
   // UNICODE_TO_GBK[30659] := 16#CD9F;
   // UNICODE_TO_GBK[30660] := 16#8715;
   // UNICODE_TO_GBK[30661] := 16#CDC9;
   // UNICODE_TO_GBK[30662] := 16#8716;
   // UNICODE_TO_GBK[30663] := 16#CDA0;
   // UNICODE_TO_GBK[30664] := 16#8717;
   // UNICODE_TO_GBK[30665] := 16#CECF;
   // UNICODE_TO_GBK[30666] := 16#8718;
   // UNICODE_TO_GBK[30667] := 16#D6A9;
   // UNICODE_TO_GBK[30668] := 16#8719;
   // UNICODE_TO_GBK[30669] := 16#CE40;
   // UNICODE_TO_GBK[30670] := 16#871A;
   // UNICODE_TO_GBK[30671] := 16#F2E3;
   // UNICODE_TO_GBK[30672] := 16#871B;
   // UNICODE_TO_GBK[30673] := 16#CE41;
   // UNICODE_TO_GBK[30674] := 16#871C;
   // UNICODE_TO_GBK[30675] := 16#C3DB;
   // UNICODE_TO_GBK[30676] := 16#871D;
   // UNICODE_TO_GBK[30677] := 16#CE42;
   // UNICODE_TO_GBK[30678] := 16#871E;
   // UNICODE_TO_GBK[30679] := 16#F2E0;
   // UNICODE_TO_GBK[30680] := 16#871F;
   // UNICODE_TO_GBK[30681] := 16#CE43;
   // UNICODE_TO_GBK[30682] := 16#8720;
   // UNICODE_TO_GBK[30683] := 16#CE44;
   // UNICODE_TO_GBK[30684] := 16#8721;
   // UNICODE_TO_GBK[30685] := 16#C0AF;
   // UNICODE_TO_GBK[30686] := 16#8722;
   // UNICODE_TO_GBK[30687] := 16#F2EC;
   // UNICODE_TO_GBK[30688] := 16#8723;
   // UNICODE_TO_GBK[30689] := 16#F2DE;
   // UNICODE_TO_GBK[30690] := 16#8724;
   // UNICODE_TO_GBK[30691] := 16#CE45;
   // UNICODE_TO_GBK[30692] := 16#8725;
   // UNICODE_TO_GBK[30693] := 16#F2E1;
   // UNICODE_TO_GBK[30694] := 16#8726;
   // UNICODE_TO_GBK[30695] := 16#CE46;
   // UNICODE_TO_GBK[30696] := 16#8727;
   // UNICODE_TO_GBK[30697] := 16#CE47;
   // UNICODE_TO_GBK[30698] := 16#8728;
   // UNICODE_TO_GBK[30699] := 16#CE48;
   // UNICODE_TO_GBK[30700] := 16#8729;
   // UNICODE_TO_GBK[30701] := 16#F2E8;
   // UNICODE_TO_GBK[30702] := 16#872A;
   // UNICODE_TO_GBK[30703] := 16#CE49;
   // UNICODE_TO_GBK[30704] := 16#872B;
   // UNICODE_TO_GBK[30705] := 16#CE4A;
   // UNICODE_TO_GBK[30706] := 16#872C;
   // UNICODE_TO_GBK[30707] := 16#CE4B;
   // UNICODE_TO_GBK[30708] := 16#872D;
   // UNICODE_TO_GBK[30709] := 16#CE4C;
   // UNICODE_TO_GBK[30710] := 16#872E;
   // UNICODE_TO_GBK[30711] := 16#F2E2;
   // UNICODE_TO_GBK[30712] := 16#872F;
   // UNICODE_TO_GBK[30713] := 16#CE4D;
   // UNICODE_TO_GBK[30714] := 16#8730;
   // UNICODE_TO_GBK[30715] := 16#CE4E;
   // UNICODE_TO_GBK[30716] := 16#8731;
   // UNICODE_TO_GBK[30717] := 16#F2E7;
   // UNICODE_TO_GBK[30718] := 16#8732;
   // UNICODE_TO_GBK[30719] := 16#CE4F;
   // UNICODE_TO_GBK[30720] := 16#8733;
   // UNICODE_TO_GBK[30721] := 16#CE50;
   // UNICODE_TO_GBK[30722] := 16#8734;
   // UNICODE_TO_GBK[30723] := 16#F2E6;
   // UNICODE_TO_GBK[30724] := 16#8735;
   // UNICODE_TO_GBK[30725] := 16#CE51;
   // UNICODE_TO_GBK[30726] := 16#8736;
   // UNICODE_TO_GBK[30727] := 16#CE52;
   // UNICODE_TO_GBK[30728] := 16#8737;
   // UNICODE_TO_GBK[30729] := 16#F2E9;
   // UNICODE_TO_GBK[30730] := 16#8738;
   // UNICODE_TO_GBK[30731] := 16#CE53;
   // UNICODE_TO_GBK[30732] := 16#8739;
   // UNICODE_TO_GBK[30733] := 16#CE54;
   // UNICODE_TO_GBK[30734] := 16#873A;
   // UNICODE_TO_GBK[30735] := 16#CE55;
   // UNICODE_TO_GBK[30736] := 16#873B;
   // UNICODE_TO_GBK[30737] := 16#F2DF;
   // UNICODE_TO_GBK[30738] := 16#873C;
   // UNICODE_TO_GBK[30739] := 16#CE56;
   // UNICODE_TO_GBK[30740] := 16#873D;
   // UNICODE_TO_GBK[30741] := 16#CE57;
   // UNICODE_TO_GBK[30742] := 16#873E;
   // UNICODE_TO_GBK[30743] := 16#F2E4;
   // UNICODE_TO_GBK[30744] := 16#873F;
   // UNICODE_TO_GBK[30745] := 16#F2EA;
   // UNICODE_TO_GBK[30746] := 16#8740;
   // UNICODE_TO_GBK[30747] := 16#CE58;
   // UNICODE_TO_GBK[30748] := 16#8741;
   // UNICODE_TO_GBK[30749] := 16#CE59;
   // UNICODE_TO_GBK[30750] := 16#8742;
   // UNICODE_TO_GBK[30751] := 16#CE5A;
   // UNICODE_TO_GBK[30752] := 16#8743;
   // UNICODE_TO_GBK[30753] := 16#CE5B;
   // UNICODE_TO_GBK[30754] := 16#8744;
   // UNICODE_TO_GBK[30755] := 16#CE5C;
   // UNICODE_TO_GBK[30756] := 16#8745;
   // UNICODE_TO_GBK[30757] := 16#CE5D;
   // UNICODE_TO_GBK[30758] := 16#8746;
   // UNICODE_TO_GBK[30759] := 16#CE5E;
   // UNICODE_TO_GBK[30760] := 16#8747;
   // UNICODE_TO_GBK[30761] := 16#D3AC;
   // UNICODE_TO_GBK[30762] := 16#8748;
   // UNICODE_TO_GBK[30763] := 16#F2E5;
   // UNICODE_TO_GBK[30764] := 16#8749;
   // UNICODE_TO_GBK[30765] := 16#B2F5;
   // UNICODE_TO_GBK[30766] := 16#874A;
   // UNICODE_TO_GBK[30767] := 16#CE5F;
   // UNICODE_TO_GBK[30768] := 16#874B;
   // UNICODE_TO_GBK[30769] := 16#CE60;
   // UNICODE_TO_GBK[30770] := 16#874C;
   // UNICODE_TO_GBK[30771] := 16#F2F2;
   // UNICODE_TO_GBK[30772] := 16#874D;
   // UNICODE_TO_GBK[30773] := 16#CE61;
   // UNICODE_TO_GBK[30774] := 16#874E;
   // UNICODE_TO_GBK[30775] := 16#D0AB;
   // UNICODE_TO_GBK[30776] := 16#874F;
   // UNICODE_TO_GBK[30777] := 16#CE62;
   // UNICODE_TO_GBK[30778] := 16#8750;
   // UNICODE_TO_GBK[30779] := 16#CE63;
   // UNICODE_TO_GBK[30780] := 16#8751;
   // UNICODE_TO_GBK[30781] := 16#CE64;
   // UNICODE_TO_GBK[30782] := 16#8752;
   // UNICODE_TO_GBK[30783] := 16#CE65;
   // UNICODE_TO_GBK[30784] := 16#8753;
   // UNICODE_TO_GBK[30785] := 16#F2F5;
   // UNICODE_TO_GBK[30786] := 16#8754;
   // UNICODE_TO_GBK[30787] := 16#CE66;
   // UNICODE_TO_GBK[30788] := 16#8755;
   // UNICODE_TO_GBK[30789] := 16#CE67;
   // UNICODE_TO_GBK[30790] := 16#8756;
   // UNICODE_TO_GBK[30791] := 16#CE68;
   // UNICODE_TO_GBK[30792] := 16#8757;
   // UNICODE_TO_GBK[30793] := 16#BBC8;
   // UNICODE_TO_GBK[30794] := 16#8758;
   // UNICODE_TO_GBK[30795] := 16#CE69;
   // UNICODE_TO_GBK[30796] := 16#8759;
   // UNICODE_TO_GBK[30797] := 16#F2F9;
   // UNICODE_TO_GBK[30798] := 16#875A;
   // UNICODE_TO_GBK[30799] := 16#CE6A;
   // UNICODE_TO_GBK[30800] := 16#875B;
   // UNICODE_TO_GBK[30801] := 16#CE6B;
   // UNICODE_TO_GBK[30802] := 16#875C;
   // UNICODE_TO_GBK[30803] := 16#CE6C;
   // UNICODE_TO_GBK[30804] := 16#875D;
   // UNICODE_TO_GBK[30805] := 16#CE6D;
   // UNICODE_TO_GBK[30806] := 16#875E;
   // UNICODE_TO_GBK[30807] := 16#CE6E;
   // UNICODE_TO_GBK[30808] := 16#875F;
   // UNICODE_TO_GBK[30809] := 16#CE6F;
   // UNICODE_TO_GBK[30810] := 16#8760;
   // UNICODE_TO_GBK[30811] := 16#F2F0;
   // UNICODE_TO_GBK[30812] := 16#8761;
   // UNICODE_TO_GBK[30813] := 16#CE70;
   // UNICODE_TO_GBK[30814] := 16#8762;
   // UNICODE_TO_GBK[30815] := 16#CE71;
   // UNICODE_TO_GBK[30816] := 16#8763;
   // UNICODE_TO_GBK[30817] := 16#F2F6;
   // UNICODE_TO_GBK[30818] := 16#8764;
   // UNICODE_TO_GBK[30819] := 16#F2F8;
   // UNICODE_TO_GBK[30820] := 16#8765;
   // UNICODE_TO_GBK[30821] := 16#F2FA;
   // UNICODE_TO_GBK[30822] := 16#8766;
   // UNICODE_TO_GBK[30823] := 16#CE72;
   // UNICODE_TO_GBK[30824] := 16#8767;
   // UNICODE_TO_GBK[30825] := 16#CE73;
   // UNICODE_TO_GBK[30826] := 16#8768;
   // UNICODE_TO_GBK[30827] := 16#CE74;
   // UNICODE_TO_GBK[30828] := 16#8769;
   // UNICODE_TO_GBK[30829] := 16#CE75;
   // UNICODE_TO_GBK[30830] := 16#876A;
   // UNICODE_TO_GBK[30831] := 16#CE76;
   // UNICODE_TO_GBK[30832] := 16#876B;
   // UNICODE_TO_GBK[30833] := 16#CE77;
   // UNICODE_TO_GBK[30834] := 16#876C;
   // UNICODE_TO_GBK[30835] := 16#CE78;
   // UNICODE_TO_GBK[30836] := 16#876D;
   // UNICODE_TO_GBK[30837] := 16#CE79;
   // UNICODE_TO_GBK[30838] := 16#876E;
   // UNICODE_TO_GBK[30839] := 16#F2F3;
   // UNICODE_TO_GBK[30840] := 16#876F;
   // UNICODE_TO_GBK[30841] := 16#CE7A;
   // UNICODE_TO_GBK[30842] := 16#8770;
   // UNICODE_TO_GBK[30843] := 16#F2F1;
   // UNICODE_TO_GBK[30844] := 16#8771;
   // UNICODE_TO_GBK[30845] := 16#CE7B;
   // UNICODE_TO_GBK[30846] := 16#8772;
   // UNICODE_TO_GBK[30847] := 16#CE7C;
   // UNICODE_TO_GBK[30848] := 16#8773;
   // UNICODE_TO_GBK[30849] := 16#CE7D;
   // UNICODE_TO_GBK[30850] := 16#8774;
   // UNICODE_TO_GBK[30851] := 16#BAFB;
   // UNICODE_TO_GBK[30852] := 16#8775;
   // UNICODE_TO_GBK[30853] := 16#CE7E;
   // UNICODE_TO_GBK[30854] := 16#8776;
   // UNICODE_TO_GBK[30855] := 16#B5FB;
   // UNICODE_TO_GBK[30856] := 16#8777;
   // UNICODE_TO_GBK[30857] := 16#CE80;
   // UNICODE_TO_GBK[30858] := 16#8778;
   // UNICODE_TO_GBK[30859] := 16#CE81;
   // UNICODE_TO_GBK[30860] := 16#8779;
   // UNICODE_TO_GBK[30861] := 16#CE82;
   // UNICODE_TO_GBK[30862] := 16#877A;
   // UNICODE_TO_GBK[30863] := 16#CE83;
   // UNICODE_TO_GBK[30864] := 16#877B;
   // UNICODE_TO_GBK[30865] := 16#F2EF;
   // UNICODE_TO_GBK[30866] := 16#877C;
   // UNICODE_TO_GBK[30867] := 16#F2F7;
   // UNICODE_TO_GBK[30868] := 16#877D;
   // UNICODE_TO_GBK[30869] := 16#F2ED;
   // UNICODE_TO_GBK[30870] := 16#877E;
   // UNICODE_TO_GBK[30871] := 16#F2EE;
   // UNICODE_TO_GBK[30872] := 16#877F;
   // UNICODE_TO_GBK[30873] := 16#CE84;
   // UNICODE_TO_GBK[30874] := 16#8780;
   // UNICODE_TO_GBK[30875] := 16#CE85;
   // UNICODE_TO_GBK[30876] := 16#8781;
   // UNICODE_TO_GBK[30877] := 16#CE86;
   // UNICODE_TO_GBK[30878] := 16#8782;
   // UNICODE_TO_GBK[30879] := 16#F2EB;
   // UNICODE_TO_GBK[30880] := 16#8783;
   // UNICODE_TO_GBK[30881] := 16#F3A6;
   // UNICODE_TO_GBK[30882] := 16#8784;
   // UNICODE_TO_GBK[30883] := 16#CE87;
   // UNICODE_TO_GBK[30884] := 16#8785;
   // UNICODE_TO_GBK[30885] := 16#F3A3;
   // UNICODE_TO_GBK[30886] := 16#8786;
   // UNICODE_TO_GBK[30887] := 16#CE88;
   // UNICODE_TO_GBK[30888] := 16#8787;
   // UNICODE_TO_GBK[30889] := 16#CE89;
   // UNICODE_TO_GBK[30890] := 16#8788;
   // UNICODE_TO_GBK[30891] := 16#F3A2;
   // UNICODE_TO_GBK[30892] := 16#8789;
   // UNICODE_TO_GBK[30893] := 16#CE8A;
   // UNICODE_TO_GBK[30894] := 16#878A;
   // UNICODE_TO_GBK[30895] := 16#CE8B;
   // UNICODE_TO_GBK[30896] := 16#878B;
   // UNICODE_TO_GBK[30897] := 16#F2F4;
   // UNICODE_TO_GBK[30898] := 16#878C;
   // UNICODE_TO_GBK[30899] := 16#CE8C;
   // UNICODE_TO_GBK[30900] := 16#878D;
   // UNICODE_TO_GBK[30901] := 16#C8DA;
   // UNICODE_TO_GBK[30902] := 16#878E;
   // UNICODE_TO_GBK[30903] := 16#CE8D;
   // UNICODE_TO_GBK[30904] := 16#878F;
   // UNICODE_TO_GBK[30905] := 16#CE8E;
   // UNICODE_TO_GBK[30906] := 16#8790;
   // UNICODE_TO_GBK[30907] := 16#CE8F;
   // UNICODE_TO_GBK[30908] := 16#8791;
   // UNICODE_TO_GBK[30909] := 16#CE90;
   // UNICODE_TO_GBK[30910] := 16#8792;
   // UNICODE_TO_GBK[30911] := 16#CE91;
   // UNICODE_TO_GBK[30912] := 16#8793;
   // UNICODE_TO_GBK[30913] := 16#F2FB;
   // UNICODE_TO_GBK[30914] := 16#8794;
   // UNICODE_TO_GBK[30915] := 16#CE92;
   // UNICODE_TO_GBK[30916] := 16#8795;
   // UNICODE_TO_GBK[30917] := 16#CE93;
   // UNICODE_TO_GBK[30918] := 16#8796;
   // UNICODE_TO_GBK[30919] := 16#CE94;
   // UNICODE_TO_GBK[30920] := 16#8797;
   // UNICODE_TO_GBK[30921] := 16#F3A5;
   // UNICODE_TO_GBK[30922] := 16#8798;
   // UNICODE_TO_GBK[30923] := 16#CE95;
   // UNICODE_TO_GBK[30924] := 16#8799;
   // UNICODE_TO_GBK[30925] := 16#CE96;
   // UNICODE_TO_GBK[30926] := 16#879A;
   // UNICODE_TO_GBK[30927] := 16#CE97;
   // UNICODE_TO_GBK[30928] := 16#879B;
   // UNICODE_TO_GBK[30929] := 16#CE98;
   // UNICODE_TO_GBK[30930] := 16#879C;
   // UNICODE_TO_GBK[30931] := 16#CE99;
   // UNICODE_TO_GBK[30932] := 16#879D;
   // UNICODE_TO_GBK[30933] := 16#CE9A;
   // UNICODE_TO_GBK[30934] := 16#879E;
   // UNICODE_TO_GBK[30935] := 16#CE9B;
   // UNICODE_TO_GBK[30936] := 16#879F;
   // UNICODE_TO_GBK[30937] := 16#C3F8;
   // UNICODE_TO_GBK[30938] := 16#87A0;
   // UNICODE_TO_GBK[30939] := 16#CE9C;
   // UNICODE_TO_GBK[30940] := 16#87A1;
   // UNICODE_TO_GBK[30941] := 16#CE9D;
   // UNICODE_TO_GBK[30942] := 16#87A2;
   // UNICODE_TO_GBK[30943] := 16#CE9E;
   // UNICODE_TO_GBK[30944] := 16#87A3;
   // UNICODE_TO_GBK[30945] := 16#CE9F;
   // UNICODE_TO_GBK[30946] := 16#87A4;
   // UNICODE_TO_GBK[30947] := 16#CEA0;
   // UNICODE_TO_GBK[30948] := 16#87A5;
   // UNICODE_TO_GBK[30949] := 16#CF40;
   // UNICODE_TO_GBK[30950] := 16#87A6;
   // UNICODE_TO_GBK[30951] := 16#CF41;
   // UNICODE_TO_GBK[30952] := 16#87A7;
   // UNICODE_TO_GBK[30953] := 16#CF42;
   // UNICODE_TO_GBK[30954] := 16#87A8;
   // UNICODE_TO_GBK[30955] := 16#F2FD;
   // UNICODE_TO_GBK[30956] := 16#87A9;
   // UNICODE_TO_GBK[30957] := 16#CF43;
   // UNICODE_TO_GBK[30958] := 16#87AA;
   // UNICODE_TO_GBK[30959] := 16#CF44;
   // UNICODE_TO_GBK[30960] := 16#87AB;
   // UNICODE_TO_GBK[30961] := 16#F3A7;
   // UNICODE_TO_GBK[30962] := 16#87AC;
   // UNICODE_TO_GBK[30963] := 16#F3A9;
   // UNICODE_TO_GBK[30964] := 16#87AD;
   // UNICODE_TO_GBK[30965] := 16#F3A4;
   // UNICODE_TO_GBK[30966] := 16#87AE;
   // UNICODE_TO_GBK[30967] := 16#CF45;
   // UNICODE_TO_GBK[30968] := 16#87AF;
   // UNICODE_TO_GBK[30969] := 16#F2FC;
   // UNICODE_TO_GBK[30970] := 16#87B0;
   // UNICODE_TO_GBK[30971] := 16#CF46;
   // UNICODE_TO_GBK[30972] := 16#87B1;
   // UNICODE_TO_GBK[30973] := 16#CF47;
   // UNICODE_TO_GBK[30974] := 16#87B2;
   // UNICODE_TO_GBK[30975] := 16#CF48;
   // UNICODE_TO_GBK[30976] := 16#87B3;
   // UNICODE_TO_GBK[30977] := 16#F3AB;
   // UNICODE_TO_GBK[30978] := 16#87B4;
   // UNICODE_TO_GBK[30979] := 16#CF49;
   // UNICODE_TO_GBK[30980] := 16#87B5;
   // UNICODE_TO_GBK[30981] := 16#F3AA;
   // UNICODE_TO_GBK[30982] := 16#87B6;
   // UNICODE_TO_GBK[30983] := 16#CF4A;
   // UNICODE_TO_GBK[30984] := 16#87B7;
   // UNICODE_TO_GBK[30985] := 16#CF4B;
   // UNICODE_TO_GBK[30986] := 16#87B8;
   // UNICODE_TO_GBK[30987] := 16#CF4C;
   // UNICODE_TO_GBK[30988] := 16#87B9;
   // UNICODE_TO_GBK[30989] := 16#CF4D;
   // UNICODE_TO_GBK[30990] := 16#87BA;
   // UNICODE_TO_GBK[30991] := 16#C2DD;
   // UNICODE_TO_GBK[30992] := 16#87BB;
   // UNICODE_TO_GBK[30993] := 16#CF4E;
   // UNICODE_TO_GBK[30994] := 16#87BC;
   // UNICODE_TO_GBK[30995] := 16#CF4F;
   // UNICODE_TO_GBK[30996] := 16#87BD;
   // UNICODE_TO_GBK[30997] := 16#F3AE;
   // UNICODE_TO_GBK[30998] := 16#87BE;
   // UNICODE_TO_GBK[30999] := 16#CF50;
   // UNICODE_TO_GBK[31000] := 16#87BF;
   // UNICODE_TO_GBK[31001] := 16#CF51;
   // UNICODE_TO_GBK[31002] := 16#87C0;
   // UNICODE_TO_GBK[31003] := 16#F3B0;
   // UNICODE_TO_GBK[31004] := 16#87C1;
   // UNICODE_TO_GBK[31005] := 16#CF52;
   // UNICODE_TO_GBK[31006] := 16#87C2;
   // UNICODE_TO_GBK[31007] := 16#CF53;
   // UNICODE_TO_GBK[31008] := 16#87C3;
   // UNICODE_TO_GBK[31009] := 16#CF54;
   // UNICODE_TO_GBK[31010] := 16#87C4;
   // UNICODE_TO_GBK[31011] := 16#CF55;
   // UNICODE_TO_GBK[31012] := 16#87C5;
   // UNICODE_TO_GBK[31013] := 16#CF56;
   // UNICODE_TO_GBK[31014] := 16#87C6;
   // UNICODE_TO_GBK[31015] := 16#F3A1;
   // UNICODE_TO_GBK[31016] := 16#87C7;
   // UNICODE_TO_GBK[31017] := 16#CF57;
   // UNICODE_TO_GBK[31018] := 16#87C8;
   // UNICODE_TO_GBK[31019] := 16#CF58;
   // UNICODE_TO_GBK[31020] := 16#87C9;
   // UNICODE_TO_GBK[31021] := 16#CF59;
   // UNICODE_TO_GBK[31022] := 16#87CA;
   // UNICODE_TO_GBK[31023] := 16#F3B1;
   // UNICODE_TO_GBK[31024] := 16#87CB;
   // UNICODE_TO_GBK[31025] := 16#F3AC;
   // UNICODE_TO_GBK[31026] := 16#87CC;
   // UNICODE_TO_GBK[31027] := 16#CF5A;
   // UNICODE_TO_GBK[31028] := 16#87CD;
   // UNICODE_TO_GBK[31029] := 16#CF5B;
   // UNICODE_TO_GBK[31030] := 16#87CE;
   // UNICODE_TO_GBK[31031] := 16#CF5C;
   // UNICODE_TO_GBK[31032] := 16#87CF;
   // UNICODE_TO_GBK[31033] := 16#CF5D;
   // UNICODE_TO_GBK[31034] := 16#87D0;
   // UNICODE_TO_GBK[31035] := 16#CF5E;
   // UNICODE_TO_GBK[31036] := 16#87D1;
   // UNICODE_TO_GBK[31037] := 16#F3AF;
   // UNICODE_TO_GBK[31038] := 16#87D2;
   // UNICODE_TO_GBK[31039] := 16#F2FE;
   // UNICODE_TO_GBK[31040] := 16#87D3;
   // UNICODE_TO_GBK[31041] := 16#F3AD;
   // UNICODE_TO_GBK[31042] := 16#87D4;
   // UNICODE_TO_GBK[31043] := 16#CF5F;
   // UNICODE_TO_GBK[31044] := 16#87D5;
   // UNICODE_TO_GBK[31045] := 16#CF60;
   // UNICODE_TO_GBK[31046] := 16#87D6;
   // UNICODE_TO_GBK[31047] := 16#CF61;
   // UNICODE_TO_GBK[31048] := 16#87D7;
   // UNICODE_TO_GBK[31049] := 16#CF62;
   // UNICODE_TO_GBK[31050] := 16#87D8;
   // UNICODE_TO_GBK[31051] := 16#CF63;
   // UNICODE_TO_GBK[31052] := 16#87D9;
   // UNICODE_TO_GBK[31053] := 16#CF64;
   // UNICODE_TO_GBK[31054] := 16#87DA;
   // UNICODE_TO_GBK[31055] := 16#CF65;
   // UNICODE_TO_GBK[31056] := 16#87DB;
   // UNICODE_TO_GBK[31057] := 16#F3B2;
   // UNICODE_TO_GBK[31058] := 16#87DC;
   // UNICODE_TO_GBK[31059] := 16#CF66;
   // UNICODE_TO_GBK[31060] := 16#87DD;
   // UNICODE_TO_GBK[31061] := 16#CF67;
   // UNICODE_TO_GBK[31062] := 16#87DE;
   // UNICODE_TO_GBK[31063] := 16#CF68;
   // UNICODE_TO_GBK[31064] := 16#87DF;
   // UNICODE_TO_GBK[31065] := 16#CF69;
   // UNICODE_TO_GBK[31066] := 16#87E0;
   // UNICODE_TO_GBK[31067] := 16#F3B4;
   // UNICODE_TO_GBK[31068] := 16#87E1;
   // UNICODE_TO_GBK[31069] := 16#CF6A;
   // UNICODE_TO_GBK[31070] := 16#87E2;
   // UNICODE_TO_GBK[31071] := 16#CF6B;
   // UNICODE_TO_GBK[31072] := 16#87E3;
   // UNICODE_TO_GBK[31073] := 16#CF6C;
   // UNICODE_TO_GBK[31074] := 16#87E4;
   // UNICODE_TO_GBK[31075] := 16#CF6D;
   // UNICODE_TO_GBK[31076] := 16#87E5;
   // UNICODE_TO_GBK[31077] := 16#F3A8;
   // UNICODE_TO_GBK[31078] := 16#87E6;
   // UNICODE_TO_GBK[31079] := 16#CF6E;
   // UNICODE_TO_GBK[31080] := 16#87E7;
   // UNICODE_TO_GBK[31081] := 16#CF6F;
   // UNICODE_TO_GBK[31082] := 16#87E8;
   // UNICODE_TO_GBK[31083] := 16#CF70;
   // UNICODE_TO_GBK[31084] := 16#87E9;
   // UNICODE_TO_GBK[31085] := 16#CF71;
   // UNICODE_TO_GBK[31086] := 16#87EA;
   // UNICODE_TO_GBK[31087] := 16#F3B3;
   // UNICODE_TO_GBK[31088] := 16#87EB;
   // UNICODE_TO_GBK[31089] := 16#CF72;
   // UNICODE_TO_GBK[31090] := 16#87EC;
   // UNICODE_TO_GBK[31091] := 16#CF73;
   // UNICODE_TO_GBK[31092] := 16#87ED;
   // UNICODE_TO_GBK[31093] := 16#CF74;
   // UNICODE_TO_GBK[31094] := 16#87EE;
   // UNICODE_TO_GBK[31095] := 16#F3B5;
   // UNICODE_TO_GBK[31096] := 16#87EF;
   // UNICODE_TO_GBK[31097] := 16#CF75;
   // UNICODE_TO_GBK[31098] := 16#87F0;
   // UNICODE_TO_GBK[31099] := 16#CF76;
   // UNICODE_TO_GBK[31100] := 16#87F1;
   // UNICODE_TO_GBK[31101] := 16#CF77;
   // UNICODE_TO_GBK[31102] := 16#87F2;
   // UNICODE_TO_GBK[31103] := 16#CF78;
   // UNICODE_TO_GBK[31104] := 16#87F3;
   // UNICODE_TO_GBK[31105] := 16#CF79;
   // UNICODE_TO_GBK[31106] := 16#87F4;
   // UNICODE_TO_GBK[31107] := 16#CF7A;
   // UNICODE_TO_GBK[31108] := 16#87F5;
   // UNICODE_TO_GBK[31109] := 16#CF7B;
   // UNICODE_TO_GBK[31110] := 16#87F6;
   // UNICODE_TO_GBK[31111] := 16#CF7C;
   // UNICODE_TO_GBK[31112] := 16#87F7;
   // UNICODE_TO_GBK[31113] := 16#CF7D;
   // UNICODE_TO_GBK[31114] := 16#87F8;
   // UNICODE_TO_GBK[31115] := 16#CF7E;
   // UNICODE_TO_GBK[31116] := 16#87F9;
   // UNICODE_TO_GBK[31117] := 16#D0B7;
   // UNICODE_TO_GBK[31118] := 16#87FA;
   // UNICODE_TO_GBK[31119] := 16#CF80;
   // UNICODE_TO_GBK[31120] := 16#87FB;
   // UNICODE_TO_GBK[31121] := 16#CF81;
   // UNICODE_TO_GBK[31122] := 16#87FC;
   // UNICODE_TO_GBK[31123] := 16#CF82;
   // UNICODE_TO_GBK[31124] := 16#87FD;
   // UNICODE_TO_GBK[31125] := 16#CF83;
   // UNICODE_TO_GBK[31126] := 16#87FE;
   // UNICODE_TO_GBK[31127] := 16#F3B8;
   // UNICODE_TO_GBK[31128] := 16#87FF;
   // UNICODE_TO_GBK[31129] := 16#CF84;
   // UNICODE_TO_GBK[31130] := 16#8800;
   // UNICODE_TO_GBK[31131] := 16#CF85;
   // UNICODE_TO_GBK[31132] := 16#8801;
   // UNICODE_TO_GBK[31133] := 16#CF86;
   // UNICODE_TO_GBK[31134] := 16#8802;
   // UNICODE_TO_GBK[31135] := 16#CF87;
   // UNICODE_TO_GBK[31136] := 16#8803;
   // UNICODE_TO_GBK[31137] := 16#D9F9;
   // UNICODE_TO_GBK[31138] := 16#8804;
   // UNICODE_TO_GBK[31139] := 16#CF88;
   // UNICODE_TO_GBK[31140] := 16#8805;
   // UNICODE_TO_GBK[31141] := 16#CF89;
   // UNICODE_TO_GBK[31142] := 16#8806;
   // UNICODE_TO_GBK[31143] := 16#CF8A;
   // UNICODE_TO_GBK[31144] := 16#8807;
   // UNICODE_TO_GBK[31145] := 16#CF8B;
   // UNICODE_TO_GBK[31146] := 16#8808;
   // UNICODE_TO_GBK[31147] := 16#CF8C;
   // UNICODE_TO_GBK[31148] := 16#8809;
   // UNICODE_TO_GBK[31149] := 16#CF8D;
   // UNICODE_TO_GBK[31150] := 16#880A;
   // UNICODE_TO_GBK[31151] := 16#F3B9;
   // UNICODE_TO_GBK[31152] := 16#880B;
   // UNICODE_TO_GBK[31153] := 16#CF8E;
   // UNICODE_TO_GBK[31154] := 16#880C;
   // UNICODE_TO_GBK[31155] := 16#CF8F;
   // UNICODE_TO_GBK[31156] := 16#880D;
   // UNICODE_TO_GBK[31157] := 16#CF90;
   // UNICODE_TO_GBK[31158] := 16#880E;
   // UNICODE_TO_GBK[31159] := 16#CF91;
   // UNICODE_TO_GBK[31160] := 16#880F;
   // UNICODE_TO_GBK[31161] := 16#CF92;
   // UNICODE_TO_GBK[31162] := 16#8810;
   // UNICODE_TO_GBK[31163] := 16#CF93;
   // UNICODE_TO_GBK[31164] := 16#8811;
   // UNICODE_TO_GBK[31165] := 16#CF94;
   // UNICODE_TO_GBK[31166] := 16#8812;
   // UNICODE_TO_GBK[31167] := 16#CF95;
   // UNICODE_TO_GBK[31168] := 16#8813;
   // UNICODE_TO_GBK[31169] := 16#F3B7;
   // UNICODE_TO_GBK[31170] := 16#8814;
   // UNICODE_TO_GBK[31171] := 16#CF96;
   // UNICODE_TO_GBK[31172] := 16#8815;
   // UNICODE_TO_GBK[31173] := 16#C8E4;
   // UNICODE_TO_GBK[31174] := 16#8816;
   // UNICODE_TO_GBK[31175] := 16#F3B6;
   // UNICODE_TO_GBK[31176] := 16#8817;
   // UNICODE_TO_GBK[31177] := 16#CF97;
   // UNICODE_TO_GBK[31178] := 16#8818;
   // UNICODE_TO_GBK[31179] := 16#CF98;
   // UNICODE_TO_GBK[31180] := 16#8819;
   // UNICODE_TO_GBK[31181] := 16#CF99;
   // UNICODE_TO_GBK[31182] := 16#881A;
   // UNICODE_TO_GBK[31183] := 16#CF9A;
   // UNICODE_TO_GBK[31184] := 16#881B;
   // UNICODE_TO_GBK[31185] := 16#F3BA;
   // UNICODE_TO_GBK[31186] := 16#881C;
   // UNICODE_TO_GBK[31187] := 16#CF9B;
   // UNICODE_TO_GBK[31188] := 16#881D;
   // UNICODE_TO_GBK[31189] := 16#CF9C;
   // UNICODE_TO_GBK[31190] := 16#881E;
   // UNICODE_TO_GBK[31191] := 16#CF9D;
   // UNICODE_TO_GBK[31192] := 16#881F;
   // UNICODE_TO_GBK[31193] := 16#CF9E;
   // UNICODE_TO_GBK[31194] := 16#8820;
   // UNICODE_TO_GBK[31195] := 16#CF9F;
   // UNICODE_TO_GBK[31196] := 16#8821;
   // UNICODE_TO_GBK[31197] := 16#F3BB;
   // UNICODE_TO_GBK[31198] := 16#8822;
   // UNICODE_TO_GBK[31199] := 16#B4C0;
   // UNICODE_TO_GBK[31200] := 16#8823;
   // UNICODE_TO_GBK[31201] := 16#CFA0;
   // UNICODE_TO_GBK[31202] := 16#8824;
   // UNICODE_TO_GBK[31203] := 16#D040;
   // UNICODE_TO_GBK[31204] := 16#8825;
   // UNICODE_TO_GBK[31205] := 16#D041;
   // UNICODE_TO_GBK[31206] := 16#8826;
   // UNICODE_TO_GBK[31207] := 16#D042;
   // UNICODE_TO_GBK[31208] := 16#8827;
   // UNICODE_TO_GBK[31209] := 16#D043;
   // UNICODE_TO_GBK[31210] := 16#8828;
   // UNICODE_TO_GBK[31211] := 16#D044;
   // UNICODE_TO_GBK[31212] := 16#8829;
   // UNICODE_TO_GBK[31213] := 16#D045;
   // UNICODE_TO_GBK[31214] := 16#882A;
   // UNICODE_TO_GBK[31215] := 16#D046;
   // UNICODE_TO_GBK[31216] := 16#882B;
   // UNICODE_TO_GBK[31217] := 16#D047;
   // UNICODE_TO_GBK[31218] := 16#882C;
   // UNICODE_TO_GBK[31219] := 16#D048;
   // UNICODE_TO_GBK[31220] := 16#882D;
   // UNICODE_TO_GBK[31221] := 16#D049;
   // UNICODE_TO_GBK[31222] := 16#882E;
   // UNICODE_TO_GBK[31223] := 16#D04A;
   // UNICODE_TO_GBK[31224] := 16#882F;
   // UNICODE_TO_GBK[31225] := 16#D04B;
   // UNICODE_TO_GBK[31226] := 16#8830;
   // UNICODE_TO_GBK[31227] := 16#D04C;
   // UNICODE_TO_GBK[31228] := 16#8831;
   // UNICODE_TO_GBK[31229] := 16#D04D;
   // UNICODE_TO_GBK[31230] := 16#8832;
   // UNICODE_TO_GBK[31231] := 16#EEC3;
   // UNICODE_TO_GBK[31232] := 16#8833;
   // UNICODE_TO_GBK[31233] := 16#D04E;
   // UNICODE_TO_GBK[31234] := 16#8834;
   // UNICODE_TO_GBK[31235] := 16#D04F;
   // UNICODE_TO_GBK[31236] := 16#8835;
   // UNICODE_TO_GBK[31237] := 16#D050;
   // UNICODE_TO_GBK[31238] := 16#8836;
   // UNICODE_TO_GBK[31239] := 16#D051;
   // UNICODE_TO_GBK[31240] := 16#8837;
   // UNICODE_TO_GBK[31241] := 16#D052;
   // UNICODE_TO_GBK[31242] := 16#8838;
   // UNICODE_TO_GBK[31243] := 16#D053;
   // UNICODE_TO_GBK[31244] := 16#8839;
   // UNICODE_TO_GBK[31245] := 16#F3BC;
   // UNICODE_TO_GBK[31246] := 16#883A;
   // UNICODE_TO_GBK[31247] := 16#D054;
   // UNICODE_TO_GBK[31248] := 16#883B;
   // UNICODE_TO_GBK[31249] := 16#D055;
   // UNICODE_TO_GBK[31250] := 16#883C;
   // UNICODE_TO_GBK[31251] := 16#F3BD;
   // UNICODE_TO_GBK[31252] := 16#883D;
   // UNICODE_TO_GBK[31253] := 16#D056;
   // UNICODE_TO_GBK[31254] := 16#883E;
   // UNICODE_TO_GBK[31255] := 16#D057;
   // UNICODE_TO_GBK[31256] := 16#883F;
   // UNICODE_TO_GBK[31257] := 16#D058;
   // UNICODE_TO_GBK[31258] := 16#8840;
   // UNICODE_TO_GBK[31259] := 16#D1AA;
   // UNICODE_TO_GBK[31260] := 16#8841;
   // UNICODE_TO_GBK[31261] := 16#D059;
   // UNICODE_TO_GBK[31262] := 16#8842;
   // UNICODE_TO_GBK[31263] := 16#D05A;
   // UNICODE_TO_GBK[31264] := 16#8843;
   // UNICODE_TO_GBK[31265] := 16#D05B;
   // UNICODE_TO_GBK[31266] := 16#8844;
   // UNICODE_TO_GBK[31267] := 16#F4AC;
   // UNICODE_TO_GBK[31268] := 16#8845;
   // UNICODE_TO_GBK[31269] := 16#D0C6;
   // UNICODE_TO_GBK[31270] := 16#8846;
   // UNICODE_TO_GBK[31271] := 16#D05C;
   // UNICODE_TO_GBK[31272] := 16#8847;
   // UNICODE_TO_GBK[31273] := 16#D05D;
   // UNICODE_TO_GBK[31274] := 16#8848;
   // UNICODE_TO_GBK[31275] := 16#D05E;
   // UNICODE_TO_GBK[31276] := 16#8849;
   // UNICODE_TO_GBK[31277] := 16#D05F;
   // UNICODE_TO_GBK[31278] := 16#884A;
   // UNICODE_TO_GBK[31279] := 16#D060;
   // UNICODE_TO_GBK[31280] := 16#884B;
   // UNICODE_TO_GBK[31281] := 16#D061;
   // UNICODE_TO_GBK[31282] := 16#884C;
   // UNICODE_TO_GBK[31283] := 16#D0D0;
   // UNICODE_TO_GBK[31284] := 16#884D;
   // UNICODE_TO_GBK[31285] := 16#D1DC;
   // UNICODE_TO_GBK[31286] := 16#884E;
   // UNICODE_TO_GBK[31287] := 16#D062;
   // UNICODE_TO_GBK[31288] := 16#884F;
   // UNICODE_TO_GBK[31289] := 16#D063;
   // UNICODE_TO_GBK[31290] := 16#8850;
   // UNICODE_TO_GBK[31291] := 16#D064;
   // UNICODE_TO_GBK[31292] := 16#8851;
   // UNICODE_TO_GBK[31293] := 16#D065;
   // UNICODE_TO_GBK[31294] := 16#8852;
   // UNICODE_TO_GBK[31295] := 16#D066;
   // UNICODE_TO_GBK[31296] := 16#8853;
   // UNICODE_TO_GBK[31297] := 16#D067;
   // UNICODE_TO_GBK[31298] := 16#8854;
   // UNICODE_TO_GBK[31299] := 16#CFCE;
   // UNICODE_TO_GBK[31300] := 16#8855;
   // UNICODE_TO_GBK[31301] := 16#D068;
   // UNICODE_TO_GBK[31302] := 16#8856;
   // UNICODE_TO_GBK[31303] := 16#D069;
   // UNICODE_TO_GBK[31304] := 16#8857;
   // UNICODE_TO_GBK[31305] := 16#BDD6;
   // UNICODE_TO_GBK[31306] := 16#8858;
   // UNICODE_TO_GBK[31307] := 16#D06A;
   // UNICODE_TO_GBK[31308] := 16#8859;
   // UNICODE_TO_GBK[31309] := 16#D1C3;
   // UNICODE_TO_GBK[31310] := 16#885A;
   // UNICODE_TO_GBK[31311] := 16#D06B;
   // UNICODE_TO_GBK[31312] := 16#885B;
   // UNICODE_TO_GBK[31313] := 16#D06C;
   // UNICODE_TO_GBK[31314] := 16#885C;
   // UNICODE_TO_GBK[31315] := 16#D06D;
   // UNICODE_TO_GBK[31316] := 16#885D;
   // UNICODE_TO_GBK[31317] := 16#D06E;
   // UNICODE_TO_GBK[31318] := 16#885E;
   // UNICODE_TO_GBK[31319] := 16#D06F;
   // UNICODE_TO_GBK[31320] := 16#885F;
   // UNICODE_TO_GBK[31321] := 16#D070;
   // UNICODE_TO_GBK[31322] := 16#8860;
   // UNICODE_TO_GBK[31323] := 16#D071;
   // UNICODE_TO_GBK[31324] := 16#8861;
   // UNICODE_TO_GBK[31325] := 16#BAE2;
   // UNICODE_TO_GBK[31326] := 16#8862;
   // UNICODE_TO_GBK[31327] := 16#E1E9;
   // UNICODE_TO_GBK[31328] := 16#8863;
   // UNICODE_TO_GBK[31329] := 16#D2C2;
   // UNICODE_TO_GBK[31330] := 16#8864;
   // UNICODE_TO_GBK[31331] := 16#F1C2;
   // UNICODE_TO_GBK[31332] := 16#8865;
   // UNICODE_TO_GBK[31333] := 16#B2B9;
   // UNICODE_TO_GBK[31334] := 16#8866;
   // UNICODE_TO_GBK[31335] := 16#D072;
   // UNICODE_TO_GBK[31336] := 16#8867;
   // UNICODE_TO_GBK[31337] := 16#D073;
   // UNICODE_TO_GBK[31338] := 16#8868;
   // UNICODE_TO_GBK[31339] := 16#B1ED;
   // UNICODE_TO_GBK[31340] := 16#8869;
   // UNICODE_TO_GBK[31341] := 16#F1C3;
   // UNICODE_TO_GBK[31342] := 16#886A;
   // UNICODE_TO_GBK[31343] := 16#D074;
   // UNICODE_TO_GBK[31344] := 16#886B;
   // UNICODE_TO_GBK[31345] := 16#C9C0;
   // UNICODE_TO_GBK[31346] := 16#886C;
   // UNICODE_TO_GBK[31347] := 16#B3C4;
   // UNICODE_TO_GBK[31348] := 16#886D;
   // UNICODE_TO_GBK[31349] := 16#D075;
   // UNICODE_TO_GBK[31350] := 16#886E;
   // UNICODE_TO_GBK[31351] := 16#D9F2;
   // UNICODE_TO_GBK[31352] := 16#886F;
   // UNICODE_TO_GBK[31353] := 16#D076;
   // UNICODE_TO_GBK[31354] := 16#8870;
   // UNICODE_TO_GBK[31355] := 16#CBA5;
   // UNICODE_TO_GBK[31356] := 16#8871;
   // UNICODE_TO_GBK[31357] := 16#D077;
   // UNICODE_TO_GBK[31358] := 16#8872;
   // UNICODE_TO_GBK[31359] := 16#F1C4;
   // UNICODE_TO_GBK[31360] := 16#8873;
   // UNICODE_TO_GBK[31361] := 16#D078;
   // UNICODE_TO_GBK[31362] := 16#8874;
   // UNICODE_TO_GBK[31363] := 16#D079;
   // UNICODE_TO_GBK[31364] := 16#8875;
   // UNICODE_TO_GBK[31365] := 16#D07A;
   // UNICODE_TO_GBK[31366] := 16#8876;
   // UNICODE_TO_GBK[31367] := 16#D07B;
   // UNICODE_TO_GBK[31368] := 16#8877;
   // UNICODE_TO_GBK[31369] := 16#D6D4;
   // UNICODE_TO_GBK[31370] := 16#8878;
   // UNICODE_TO_GBK[31371] := 16#D07C;
   // UNICODE_TO_GBK[31372] := 16#8879;
   // UNICODE_TO_GBK[31373] := 16#D07D;
   // UNICODE_TO_GBK[31374] := 16#887A;
   // UNICODE_TO_GBK[31375] := 16#D07E;
   // UNICODE_TO_GBK[31376] := 16#887B;
   // UNICODE_TO_GBK[31377] := 16#D080;
   // UNICODE_TO_GBK[31378] := 16#887C;
   // UNICODE_TO_GBK[31379] := 16#D081;
   // UNICODE_TO_GBK[31380] := 16#887D;
   // UNICODE_TO_GBK[31381] := 16#F1C5;
   // UNICODE_TO_GBK[31382] := 16#887E;
   // UNICODE_TO_GBK[31383] := 16#F4C0;
   // UNICODE_TO_GBK[31384] := 16#887F;
   // UNICODE_TO_GBK[31385] := 16#F1C6;
   // UNICODE_TO_GBK[31386] := 16#8880;
   // UNICODE_TO_GBK[31387] := 16#D082;
   // UNICODE_TO_GBK[31388] := 16#8881;
   // UNICODE_TO_GBK[31389] := 16#D4AC;
   // UNICODE_TO_GBK[31390] := 16#8882;
   // UNICODE_TO_GBK[31391] := 16#F1C7;
   // UNICODE_TO_GBK[31392] := 16#8883;
   // UNICODE_TO_GBK[31393] := 16#D083;
   // UNICODE_TO_GBK[31394] := 16#8884;
   // UNICODE_TO_GBK[31395] := 16#B0C0;
   // UNICODE_TO_GBK[31396] := 16#8885;
   // UNICODE_TO_GBK[31397] := 16#F4C1;
   // UNICODE_TO_GBK[31398] := 16#8886;
   // UNICODE_TO_GBK[31399] := 16#D084;
   // UNICODE_TO_GBK[31400] := 16#8887;
   // UNICODE_TO_GBK[31401] := 16#D085;
   // UNICODE_TO_GBK[31402] := 16#8888;
   // UNICODE_TO_GBK[31403] := 16#F4C2;
   // UNICODE_TO_GBK[31404] := 16#8889;
   // UNICODE_TO_GBK[31405] := 16#D086;
   // UNICODE_TO_GBK[31406] := 16#888A;
   // UNICODE_TO_GBK[31407] := 16#D087;
   // UNICODE_TO_GBK[31408] := 16#888B;
   // UNICODE_TO_GBK[31409] := 16#B4FC;
   // UNICODE_TO_GBK[31410] := 16#888C;
   // UNICODE_TO_GBK[31411] := 16#D088;
   // UNICODE_TO_GBK[31412] := 16#888D;
   // UNICODE_TO_GBK[31413] := 16#C5DB;
   // UNICODE_TO_GBK[31414] := 16#888E;
   // UNICODE_TO_GBK[31415] := 16#D089;
   // UNICODE_TO_GBK[31416] := 16#888F;
   // UNICODE_TO_GBK[31417] := 16#D08A;
   // UNICODE_TO_GBK[31418] := 16#8890;
   // UNICODE_TO_GBK[31419] := 16#D08B;
   // UNICODE_TO_GBK[31420] := 16#8891;
   // UNICODE_TO_GBK[31421] := 16#D08C;
   // UNICODE_TO_GBK[31422] := 16#8892;
   // UNICODE_TO_GBK[31423] := 16#CCBB;
   // UNICODE_TO_GBK[31424] := 16#8893;
   // UNICODE_TO_GBK[31425] := 16#D08D;
   // UNICODE_TO_GBK[31426] := 16#8894;
   // UNICODE_TO_GBK[31427] := 16#D08E;
   // UNICODE_TO_GBK[31428] := 16#8895;
   // UNICODE_TO_GBK[31429] := 16#D08F;
   // UNICODE_TO_GBK[31430] := 16#8896;
   // UNICODE_TO_GBK[31431] := 16#D0E4;
   // UNICODE_TO_GBK[31432] := 16#8897;
   // UNICODE_TO_GBK[31433] := 16#D090;
   // UNICODE_TO_GBK[31434] := 16#8898;
   // UNICODE_TO_GBK[31435] := 16#D091;
   // UNICODE_TO_GBK[31436] := 16#8899;
   // UNICODE_TO_GBK[31437] := 16#D092;
   // UNICODE_TO_GBK[31438] := 16#889A;
   // UNICODE_TO_GBK[31439] := 16#D093;
   // UNICODE_TO_GBK[31440] := 16#889B;
   // UNICODE_TO_GBK[31441] := 16#D094;
   // UNICODE_TO_GBK[31442] := 16#889C;
   // UNICODE_TO_GBK[31443] := 16#CDE0;
   // UNICODE_TO_GBK[31444] := 16#889D;
   // UNICODE_TO_GBK[31445] := 16#D095;
   // UNICODE_TO_GBK[31446] := 16#889E;
   // UNICODE_TO_GBK[31447] := 16#D096;
   // UNICODE_TO_GBK[31448] := 16#889F;
   // UNICODE_TO_GBK[31449] := 16#D097;
   // UNICODE_TO_GBK[31450] := 16#88A0;
   // UNICODE_TO_GBK[31451] := 16#D098;
   // UNICODE_TO_GBK[31452] := 16#88A1;
   // UNICODE_TO_GBK[31453] := 16#D099;
   // UNICODE_TO_GBK[31454] := 16#88A2;
   // UNICODE_TO_GBK[31455] := 16#F1C8;
   // UNICODE_TO_GBK[31456] := 16#88A3;
   // UNICODE_TO_GBK[31457] := 16#D09A;
   // UNICODE_TO_GBK[31458] := 16#88A4;
   // UNICODE_TO_GBK[31459] := 16#D9F3;
   // UNICODE_TO_GBK[31460] := 16#88A5;
   // UNICODE_TO_GBK[31461] := 16#D09B;
   // UNICODE_TO_GBK[31462] := 16#88A6;
   // UNICODE_TO_GBK[31463] := 16#D09C;
   // UNICODE_TO_GBK[31464] := 16#88A7;
   // UNICODE_TO_GBK[31465] := 16#D09D;
   // UNICODE_TO_GBK[31466] := 16#88A8;
   // UNICODE_TO_GBK[31467] := 16#D09E;
   // UNICODE_TO_GBK[31468] := 16#88A9;
   // UNICODE_TO_GBK[31469] := 16#D09F;
   // UNICODE_TO_GBK[31470] := 16#88AA;
   // UNICODE_TO_GBK[31471] := 16#D0A0;
   // UNICODE_TO_GBK[31472] := 16#88AB;
   // UNICODE_TO_GBK[31473] := 16#B1BB;
   // UNICODE_TO_GBK[31474] := 16#88AC;
   // UNICODE_TO_GBK[31475] := 16#D140;
   // UNICODE_TO_GBK[31476] := 16#88AD;
   // UNICODE_TO_GBK[31477] := 16#CFAE;
   // UNICODE_TO_GBK[31478] := 16#88AE;
   // UNICODE_TO_GBK[31479] := 16#D141;
   // UNICODE_TO_GBK[31480] := 16#88AF;
   // UNICODE_TO_GBK[31481] := 16#D142;
   // UNICODE_TO_GBK[31482] := 16#88B0;
   // UNICODE_TO_GBK[31483] := 16#D143;
   // UNICODE_TO_GBK[31484] := 16#88B1;
   // UNICODE_TO_GBK[31485] := 16#B8A4;
   // UNICODE_TO_GBK[31486] := 16#88B2;
   // UNICODE_TO_GBK[31487] := 16#D144;
   // UNICODE_TO_GBK[31488] := 16#88B3;
   // UNICODE_TO_GBK[31489] := 16#D145;
   // UNICODE_TO_GBK[31490] := 16#88B4;
   // UNICODE_TO_GBK[31491] := 16#D146;
   // UNICODE_TO_GBK[31492] := 16#88B5;
   // UNICODE_TO_GBK[31493] := 16#D147;
   // UNICODE_TO_GBK[31494] := 16#88B6;
   // UNICODE_TO_GBK[31495] := 16#D148;
   // UNICODE_TO_GBK[31496] := 16#88B7;
   // UNICODE_TO_GBK[31497] := 16#F1CA;
   // UNICODE_TO_GBK[31498] := 16#88B8;
   // UNICODE_TO_GBK[31499] := 16#D149;
   // UNICODE_TO_GBK[31500] := 16#88B9;
   // UNICODE_TO_GBK[31501] := 16#D14A;
   // UNICODE_TO_GBK[31502] := 16#88BA;
   // UNICODE_TO_GBK[31503] := 16#D14B;
   // UNICODE_TO_GBK[31504] := 16#88BB;
   // UNICODE_TO_GBK[31505] := 16#D14C;
   // UNICODE_TO_GBK[31506] := 16#88BC;
   // UNICODE_TO_GBK[31507] := 16#F1CB;
   // UNICODE_TO_GBK[31508] := 16#88BD;
   // UNICODE_TO_GBK[31509] := 16#D14D;
   // UNICODE_TO_GBK[31510] := 16#88BE;
   // UNICODE_TO_GBK[31511] := 16#D14E;
   // UNICODE_TO_GBK[31512] := 16#88BF;
   // UNICODE_TO_GBK[31513] := 16#D14F;
   // UNICODE_TO_GBK[31514] := 16#88C0;
   // UNICODE_TO_GBK[31515] := 16#D150;
   // UNICODE_TO_GBK[31516] := 16#88C1;
   // UNICODE_TO_GBK[31517] := 16#B2C3;
   // UNICODE_TO_GBK[31518] := 16#88C2;
   // UNICODE_TO_GBK[31519] := 16#C1D1;
   // UNICODE_TO_GBK[31520] := 16#88C3;
   // UNICODE_TO_GBK[31521] := 16#D151;
   // UNICODE_TO_GBK[31522] := 16#88C4;
   // UNICODE_TO_GBK[31523] := 16#D152;
   // UNICODE_TO_GBK[31524] := 16#88C5;
   // UNICODE_TO_GBK[31525] := 16#D7B0;
   // UNICODE_TO_GBK[31526] := 16#88C6;
   // UNICODE_TO_GBK[31527] := 16#F1C9;
   // UNICODE_TO_GBK[31528] := 16#88C7;
   // UNICODE_TO_GBK[31529] := 16#D153;
   // UNICODE_TO_GBK[31530] := 16#88C8;
   // UNICODE_TO_GBK[31531] := 16#D154;
   // UNICODE_TO_GBK[31532] := 16#88C9;
   // UNICODE_TO_GBK[31533] := 16#F1CC;
   // UNICODE_TO_GBK[31534] := 16#88CA;
   // UNICODE_TO_GBK[31535] := 16#D155;
   // UNICODE_TO_GBK[31536] := 16#88CB;
   // UNICODE_TO_GBK[31537] := 16#D156;
   // UNICODE_TO_GBK[31538] := 16#88CC;
   // UNICODE_TO_GBK[31539] := 16#D157;
   // UNICODE_TO_GBK[31540] := 16#88CD;
   // UNICODE_TO_GBK[31541] := 16#D158;
   // UNICODE_TO_GBK[31542] := 16#88CE;
   // UNICODE_TO_GBK[31543] := 16#F1CE;
   // UNICODE_TO_GBK[31544] := 16#88CF;
   // UNICODE_TO_GBK[31545] := 16#D159;
   // UNICODE_TO_GBK[31546] := 16#88D0;
   // UNICODE_TO_GBK[31547] := 16#D15A;
   // UNICODE_TO_GBK[31548] := 16#88D1;
   // UNICODE_TO_GBK[31549] := 16#D15B;
   // UNICODE_TO_GBK[31550] := 16#88D2;
   // UNICODE_TO_GBK[31551] := 16#D9F6;
   // UNICODE_TO_GBK[31552] := 16#88D3;
   // UNICODE_TO_GBK[31553] := 16#D15C;
   // UNICODE_TO_GBK[31554] := 16#88D4;
   // UNICODE_TO_GBK[31555] := 16#D2E1;
   // UNICODE_TO_GBK[31556] := 16#88D5;
   // UNICODE_TO_GBK[31557] := 16#D4A3;
   // UNICODE_TO_GBK[31558] := 16#88D6;
   // UNICODE_TO_GBK[31559] := 16#D15D;
   // UNICODE_TO_GBK[31560] := 16#88D7;
   // UNICODE_TO_GBK[31561] := 16#D15E;
   // UNICODE_TO_GBK[31562] := 16#88D8;
   // UNICODE_TO_GBK[31563] := 16#F4C3;
   // UNICODE_TO_GBK[31564] := 16#88D9;
   // UNICODE_TO_GBK[31565] := 16#C8B9;
   // UNICODE_TO_GBK[31566] := 16#88DA;
   // UNICODE_TO_GBK[31567] := 16#D15F;
   // UNICODE_TO_GBK[31568] := 16#88DB;
   // UNICODE_TO_GBK[31569] := 16#D160;
   // UNICODE_TO_GBK[31570] := 16#88DC;
   // UNICODE_TO_GBK[31571] := 16#D161;
   // UNICODE_TO_GBK[31572] := 16#88DD;
   // UNICODE_TO_GBK[31573] := 16#D162;
   // UNICODE_TO_GBK[31574] := 16#88DE;
   // UNICODE_TO_GBK[31575] := 16#D163;
   // UNICODE_TO_GBK[31576] := 16#88DF;
   // UNICODE_TO_GBK[31577] := 16#F4C4;
   // UNICODE_TO_GBK[31578] := 16#88E0;
   // UNICODE_TO_GBK[31579] := 16#D164;
   // UNICODE_TO_GBK[31580] := 16#88E1;
   // UNICODE_TO_GBK[31581] := 16#D165;
   // UNICODE_TO_GBK[31582] := 16#88E2;
   // UNICODE_TO_GBK[31583] := 16#F1CD;
   // UNICODE_TO_GBK[31584] := 16#88E3;
   // UNICODE_TO_GBK[31585] := 16#F1CF;
   // UNICODE_TO_GBK[31586] := 16#88E4;
   // UNICODE_TO_GBK[31587] := 16#BFE3;
   // UNICODE_TO_GBK[31588] := 16#88E5;
   // UNICODE_TO_GBK[31589] := 16#F1D0;
   // UNICODE_TO_GBK[31590] := 16#88E6;
   // UNICODE_TO_GBK[31591] := 16#D166;
   // UNICODE_TO_GBK[31592] := 16#88E7;
   // UNICODE_TO_GBK[31593] := 16#D167;
   // UNICODE_TO_GBK[31594] := 16#88E8;
   // UNICODE_TO_GBK[31595] := 16#F1D4;
   // UNICODE_TO_GBK[31596] := 16#88E9;
   // UNICODE_TO_GBK[31597] := 16#D168;
   // UNICODE_TO_GBK[31598] := 16#88EA;
   // UNICODE_TO_GBK[31599] := 16#D169;
   // UNICODE_TO_GBK[31600] := 16#88EB;
   // UNICODE_TO_GBK[31601] := 16#D16A;
   // UNICODE_TO_GBK[31602] := 16#88EC;
   // UNICODE_TO_GBK[31603] := 16#D16B;
   // UNICODE_TO_GBK[31604] := 16#88ED;
   // UNICODE_TO_GBK[31605] := 16#D16C;
   // UNICODE_TO_GBK[31606] := 16#88EE;
   // UNICODE_TO_GBK[31607] := 16#D16D;
   // UNICODE_TO_GBK[31608] := 16#88EF;
   // UNICODE_TO_GBK[31609] := 16#D16E;
   // UNICODE_TO_GBK[31610] := 16#88F0;
   // UNICODE_TO_GBK[31611] := 16#F1D6;
   // UNICODE_TO_GBK[31612] := 16#88F1;
   // UNICODE_TO_GBK[31613] := 16#F1D1;
   // UNICODE_TO_GBK[31614] := 16#88F2;
   // UNICODE_TO_GBK[31615] := 16#D16F;
   // UNICODE_TO_GBK[31616] := 16#88F3;
   // UNICODE_TO_GBK[31617] := 16#C9D1;
   // UNICODE_TO_GBK[31618] := 16#88F4;
   // UNICODE_TO_GBK[31619] := 16#C5E1;
   // UNICODE_TO_GBK[31620] := 16#88F5;
   // UNICODE_TO_GBK[31621] := 16#D170;
   // UNICODE_TO_GBK[31622] := 16#88F6;
   // UNICODE_TO_GBK[31623] := 16#D171;
   // UNICODE_TO_GBK[31624] := 16#88F7;
   // UNICODE_TO_GBK[31625] := 16#D172;
   // UNICODE_TO_GBK[31626] := 16#88F8;
   // UNICODE_TO_GBK[31627] := 16#C2E3;
   // UNICODE_TO_GBK[31628] := 16#88F9;
   // UNICODE_TO_GBK[31629] := 16#B9FC;
   // UNICODE_TO_GBK[31630] := 16#88FA;
   // UNICODE_TO_GBK[31631] := 16#D173;
   // UNICODE_TO_GBK[31632] := 16#88FB;
   // UNICODE_TO_GBK[31633] := 16#D174;
   // UNICODE_TO_GBK[31634] := 16#88FC;
   // UNICODE_TO_GBK[31635] := 16#F1D3;
   // UNICODE_TO_GBK[31636] := 16#88FD;
   // UNICODE_TO_GBK[31637] := 16#D175;
   // UNICODE_TO_GBK[31638] := 16#88FE;
   // UNICODE_TO_GBK[31639] := 16#F1D5;
   // UNICODE_TO_GBK[31640] := 16#88FF;
   // UNICODE_TO_GBK[31641] := 16#D176;
   // UNICODE_TO_GBK[31642] := 16#8900;
   // UNICODE_TO_GBK[31643] := 16#D177;
   // UNICODE_TO_GBK[31644] := 16#8901;
   // UNICODE_TO_GBK[31645] := 16#D178;
   // UNICODE_TO_GBK[31646] := 16#8902;
   // UNICODE_TO_GBK[31647] := 16#B9D3;
   // UNICODE_TO_GBK[31648] := 16#8903;
   // UNICODE_TO_GBK[31649] := 16#D179;
   // UNICODE_TO_GBK[31650] := 16#8904;
   // UNICODE_TO_GBK[31651] := 16#D17A;
   // UNICODE_TO_GBK[31652] := 16#8905;
   // UNICODE_TO_GBK[31653] := 16#D17B;
   // UNICODE_TO_GBK[31654] := 16#8906;
   // UNICODE_TO_GBK[31655] := 16#D17C;
   // UNICODE_TO_GBK[31656] := 16#8907;
   // UNICODE_TO_GBK[31657] := 16#D17D;
   // UNICODE_TO_GBK[31658] := 16#8908;
   // UNICODE_TO_GBK[31659] := 16#D17E;
   // UNICODE_TO_GBK[31660] := 16#8909;
   // UNICODE_TO_GBK[31661] := 16#D180;
   // UNICODE_TO_GBK[31662] := 16#890A;
   // UNICODE_TO_GBK[31663] := 16#F1DB;
   // UNICODE_TO_GBK[31664] := 16#890B;
   // UNICODE_TO_GBK[31665] := 16#D181;
   // UNICODE_TO_GBK[31666] := 16#890C;
   // UNICODE_TO_GBK[31667] := 16#D182;
   // UNICODE_TO_GBK[31668] := 16#890D;
   // UNICODE_TO_GBK[31669] := 16#D183;
   // UNICODE_TO_GBK[31670] := 16#890E;
   // UNICODE_TO_GBK[31671] := 16#D184;
   // UNICODE_TO_GBK[31672] := 16#890F;
   // UNICODE_TO_GBK[31673] := 16#D185;
   // UNICODE_TO_GBK[31674] := 16#8910;
   // UNICODE_TO_GBK[31675] := 16#BAD6;
   // UNICODE_TO_GBK[31676] := 16#8911;
   // UNICODE_TO_GBK[31677] := 16#D186;
   // UNICODE_TO_GBK[31678] := 16#8912;
   // UNICODE_TO_GBK[31679] := 16#B0FD;
   // UNICODE_TO_GBK[31680] := 16#8913;
   // UNICODE_TO_GBK[31681] := 16#F1D9;
   // UNICODE_TO_GBK[31682] := 16#8914;
   // UNICODE_TO_GBK[31683] := 16#D187;
   // UNICODE_TO_GBK[31684] := 16#8915;
   // UNICODE_TO_GBK[31685] := 16#D188;
   // UNICODE_TO_GBK[31686] := 16#8916;
   // UNICODE_TO_GBK[31687] := 16#D189;
   // UNICODE_TO_GBK[31688] := 16#8917;
   // UNICODE_TO_GBK[31689] := 16#D18A;
   // UNICODE_TO_GBK[31690] := 16#8918;
   // UNICODE_TO_GBK[31691] := 16#D18B;
   // UNICODE_TO_GBK[31692] := 16#8919;
   // UNICODE_TO_GBK[31693] := 16#F1D8;
   // UNICODE_TO_GBK[31694] := 16#891A;
   // UNICODE_TO_GBK[31695] := 16#F1D2;
   // UNICODE_TO_GBK[31696] := 16#891B;
   // UNICODE_TO_GBK[31697] := 16#F1DA;
   // UNICODE_TO_GBK[31698] := 16#891C;
   // UNICODE_TO_GBK[31699] := 16#D18C;
   // UNICODE_TO_GBK[31700] := 16#891D;
   // UNICODE_TO_GBK[31701] := 16#D18D;
   // UNICODE_TO_GBK[31702] := 16#891E;
   // UNICODE_TO_GBK[31703] := 16#D18E;
   // UNICODE_TO_GBK[31704] := 16#891F;
   // UNICODE_TO_GBK[31705] := 16#D18F;
   // UNICODE_TO_GBK[31706] := 16#8920;
   // UNICODE_TO_GBK[31707] := 16#D190;
   // UNICODE_TO_GBK[31708] := 16#8921;
   // UNICODE_TO_GBK[31709] := 16#F1D7;
   // UNICODE_TO_GBK[31710] := 16#8922;
   // UNICODE_TO_GBK[31711] := 16#D191;
   // UNICODE_TO_GBK[31712] := 16#8923;
   // UNICODE_TO_GBK[31713] := 16#D192;
   // UNICODE_TO_GBK[31714] := 16#8924;
   // UNICODE_TO_GBK[31715] := 16#D193;
   // UNICODE_TO_GBK[31716] := 16#8925;
   // UNICODE_TO_GBK[31717] := 16#C8EC;
   // UNICODE_TO_GBK[31718] := 16#8926;
   // UNICODE_TO_GBK[31719] := 16#D194;
   // UNICODE_TO_GBK[31720] := 16#8927;
   // UNICODE_TO_GBK[31721] := 16#D195;
   // UNICODE_TO_GBK[31722] := 16#8928;
   // UNICODE_TO_GBK[31723] := 16#D196;
   // UNICODE_TO_GBK[31724] := 16#8929;
   // UNICODE_TO_GBK[31725] := 16#D197;
   // UNICODE_TO_GBK[31726] := 16#892A;
   // UNICODE_TO_GBK[31727] := 16#CDCA;
   // UNICODE_TO_GBK[31728] := 16#892B;
   // UNICODE_TO_GBK[31729] := 16#F1DD;
   // UNICODE_TO_GBK[31730] := 16#892C;
   // UNICODE_TO_GBK[31731] := 16#D198;
   // UNICODE_TO_GBK[31732] := 16#892D;
   // UNICODE_TO_GBK[31733] := 16#D199;
   // UNICODE_TO_GBK[31734] := 16#892E;
   // UNICODE_TO_GBK[31735] := 16#D19A;
   // UNICODE_TO_GBK[31736] := 16#892F;
   // UNICODE_TO_GBK[31737] := 16#D19B;
   // UNICODE_TO_GBK[31738] := 16#8930;
   // UNICODE_TO_GBK[31739] := 16#E5BD;
   // UNICODE_TO_GBK[31740] := 16#8931;
   // UNICODE_TO_GBK[31741] := 16#D19C;
   // UNICODE_TO_GBK[31742] := 16#8932;
   // UNICODE_TO_GBK[31743] := 16#D19D;
   // UNICODE_TO_GBK[31744] := 16#8933;
   // UNICODE_TO_GBK[31745] := 16#D19E;
   // UNICODE_TO_GBK[31746] := 16#8934;
   // UNICODE_TO_GBK[31747] := 16#F1DC;
   // UNICODE_TO_GBK[31748] := 16#8935;
   // UNICODE_TO_GBK[31749] := 16#D19F;
   // UNICODE_TO_GBK[31750] := 16#8936;
   // UNICODE_TO_GBK[31751] := 16#F1DE;
   // UNICODE_TO_GBK[31752] := 16#8937;
   // UNICODE_TO_GBK[31753] := 16#D1A0;
   // UNICODE_TO_GBK[31754] := 16#8938;
   // UNICODE_TO_GBK[31755] := 16#D240;
   // UNICODE_TO_GBK[31756] := 16#8939;
   // UNICODE_TO_GBK[31757] := 16#D241;
   // UNICODE_TO_GBK[31758] := 16#893A;
   // UNICODE_TO_GBK[31759] := 16#D242;
   // UNICODE_TO_GBK[31760] := 16#893B;
   // UNICODE_TO_GBK[31761] := 16#D243;
   // UNICODE_TO_GBK[31762] := 16#893C;
   // UNICODE_TO_GBK[31763] := 16#D244;
   // UNICODE_TO_GBK[31764] := 16#893D;
   // UNICODE_TO_GBK[31765] := 16#D245;
   // UNICODE_TO_GBK[31766] := 16#893E;
   // UNICODE_TO_GBK[31767] := 16#D246;
   // UNICODE_TO_GBK[31768] := 16#893F;
   // UNICODE_TO_GBK[31769] := 16#D247;
   // UNICODE_TO_GBK[31770] := 16#8940;
   // UNICODE_TO_GBK[31771] := 16#D248;
   // UNICODE_TO_GBK[31772] := 16#8941;
   // UNICODE_TO_GBK[31773] := 16#F1DF;
   // UNICODE_TO_GBK[31774] := 16#8942;
   // UNICODE_TO_GBK[31775] := 16#D249;
   // UNICODE_TO_GBK[31776] := 16#8943;
   // UNICODE_TO_GBK[31777] := 16#D24A;
   // UNICODE_TO_GBK[31778] := 16#8944;
   // UNICODE_TO_GBK[31779] := 16#CFE5;
   // UNICODE_TO_GBK[31780] := 16#8945;
   // UNICODE_TO_GBK[31781] := 16#D24B;
   // UNICODE_TO_GBK[31782] := 16#8946;
   // UNICODE_TO_GBK[31783] := 16#D24C;
   // UNICODE_TO_GBK[31784] := 16#8947;
   // UNICODE_TO_GBK[31785] := 16#D24D;
   // UNICODE_TO_GBK[31786] := 16#8948;
   // UNICODE_TO_GBK[31787] := 16#D24E;
   // UNICODE_TO_GBK[31788] := 16#8949;
   // UNICODE_TO_GBK[31789] := 16#D24F;
   // UNICODE_TO_GBK[31790] := 16#894A;
   // UNICODE_TO_GBK[31791] := 16#D250;
   // UNICODE_TO_GBK[31792] := 16#894B;
   // UNICODE_TO_GBK[31793] := 16#D251;
   // UNICODE_TO_GBK[31794] := 16#894C;
   // UNICODE_TO_GBK[31795] := 16#D252;
   // UNICODE_TO_GBK[31796] := 16#894D;
   // UNICODE_TO_GBK[31797] := 16#D253;
   // UNICODE_TO_GBK[31798] := 16#894E;
   // UNICODE_TO_GBK[31799] := 16#D254;
   // UNICODE_TO_GBK[31800] := 16#894F;
   // UNICODE_TO_GBK[31801] := 16#D255;
   // UNICODE_TO_GBK[31802] := 16#8950;
   // UNICODE_TO_GBK[31803] := 16#D256;
   // UNICODE_TO_GBK[31804] := 16#8951;
   // UNICODE_TO_GBK[31805] := 16#D257;
   // UNICODE_TO_GBK[31806] := 16#8952;
   // UNICODE_TO_GBK[31807] := 16#D258;
   // UNICODE_TO_GBK[31808] := 16#8953;
   // UNICODE_TO_GBK[31809] := 16#D259;
   // UNICODE_TO_GBK[31810] := 16#8954;
   // UNICODE_TO_GBK[31811] := 16#D25A;
   // UNICODE_TO_GBK[31812] := 16#8955;
   // UNICODE_TO_GBK[31813] := 16#D25B;
   // UNICODE_TO_GBK[31814] := 16#8956;
   // UNICODE_TO_GBK[31815] := 16#D25C;
   // UNICODE_TO_GBK[31816] := 16#8957;
   // UNICODE_TO_GBK[31817] := 16#D25D;
   // UNICODE_TO_GBK[31818] := 16#8958;
   // UNICODE_TO_GBK[31819] := 16#D25E;
   // UNICODE_TO_GBK[31820] := 16#8959;
   // UNICODE_TO_GBK[31821] := 16#D25F;
   // UNICODE_TO_GBK[31822] := 16#895A;
   // UNICODE_TO_GBK[31823] := 16#D260;
   // UNICODE_TO_GBK[31824] := 16#895B;
   // UNICODE_TO_GBK[31825] := 16#D261;
   // UNICODE_TO_GBK[31826] := 16#895C;
   // UNICODE_TO_GBK[31827] := 16#D262;
   // UNICODE_TO_GBK[31828] := 16#895D;
   // UNICODE_TO_GBK[31829] := 16#D263;
   // UNICODE_TO_GBK[31830] := 16#895E;
   // UNICODE_TO_GBK[31831] := 16#F4C5;
   // UNICODE_TO_GBK[31832] := 16#895F;
   // UNICODE_TO_GBK[31833] := 16#BDF3;
   // UNICODE_TO_GBK[31834] := 16#8960;
   // UNICODE_TO_GBK[31835] := 16#D264;
   // UNICODE_TO_GBK[31836] := 16#8961;
   // UNICODE_TO_GBK[31837] := 16#D265;
   // UNICODE_TO_GBK[31838] := 16#8962;
   // UNICODE_TO_GBK[31839] := 16#D266;
   // UNICODE_TO_GBK[31840] := 16#8963;
   // UNICODE_TO_GBK[31841] := 16#D267;
   // UNICODE_TO_GBK[31842] := 16#8964;
   // UNICODE_TO_GBK[31843] := 16#D268;
   // UNICODE_TO_GBK[31844] := 16#8965;
   // UNICODE_TO_GBK[31845] := 16#D269;
   // UNICODE_TO_GBK[31846] := 16#8966;
   // UNICODE_TO_GBK[31847] := 16#F1E0;
   // UNICODE_TO_GBK[31848] := 16#8967;
   // UNICODE_TO_GBK[31849] := 16#D26A;
   // UNICODE_TO_GBK[31850] := 16#8968;
   // UNICODE_TO_GBK[31851] := 16#D26B;
   // UNICODE_TO_GBK[31852] := 16#8969;
   // UNICODE_TO_GBK[31853] := 16#D26C;
   // UNICODE_TO_GBK[31854] := 16#896A;
   // UNICODE_TO_GBK[31855] := 16#D26D;
   // UNICODE_TO_GBK[31856] := 16#896B;
   // UNICODE_TO_GBK[31857] := 16#D26E;
   // UNICODE_TO_GBK[31858] := 16#896C;
   // UNICODE_TO_GBK[31859] := 16#D26F;
   // UNICODE_TO_GBK[31860] := 16#896D;
   // UNICODE_TO_GBK[31861] := 16#D270;
   // UNICODE_TO_GBK[31862] := 16#896E;
   // UNICODE_TO_GBK[31863] := 16#D271;
   // UNICODE_TO_GBK[31864] := 16#896F;
   // UNICODE_TO_GBK[31865] := 16#D272;
   // UNICODE_TO_GBK[31866] := 16#8970;
   // UNICODE_TO_GBK[31867] := 16#D273;
   // UNICODE_TO_GBK[31868] := 16#8971;
   // UNICODE_TO_GBK[31869] := 16#D274;
   // UNICODE_TO_GBK[31870] := 16#8972;
   // UNICODE_TO_GBK[31871] := 16#D275;
   // UNICODE_TO_GBK[31872] := 16#8973;
   // UNICODE_TO_GBK[31873] := 16#D276;
   // UNICODE_TO_GBK[31874] := 16#8974;
   // UNICODE_TO_GBK[31875] := 16#D277;
   // UNICODE_TO_GBK[31876] := 16#8975;
   // UNICODE_TO_GBK[31877] := 16#D278;
   // UNICODE_TO_GBK[31878] := 16#8976;
   // UNICODE_TO_GBK[31879] := 16#D279;
   // UNICODE_TO_GBK[31880] := 16#8977;
   // UNICODE_TO_GBK[31881] := 16#D27A;
   // UNICODE_TO_GBK[31882] := 16#8978;
   // UNICODE_TO_GBK[31883] := 16#D27B;
   // UNICODE_TO_GBK[31884] := 16#8979;
   // UNICODE_TO_GBK[31885] := 16#D27C;
   // UNICODE_TO_GBK[31886] := 16#897A;
   // UNICODE_TO_GBK[31887] := 16#D27D;
   // UNICODE_TO_GBK[31888] := 16#897B;
   // UNICODE_TO_GBK[31889] := 16#F1E1;
   // UNICODE_TO_GBK[31890] := 16#897C;
   // UNICODE_TO_GBK[31891] := 16#D27E;
   // UNICODE_TO_GBK[31892] := 16#897D;
   // UNICODE_TO_GBK[31893] := 16#D280;
   // UNICODE_TO_GBK[31894] := 16#897E;
   // UNICODE_TO_GBK[31895] := 16#D281;
   // UNICODE_TO_GBK[31896] := 16#897F;
   // UNICODE_TO_GBK[31897] := 16#CEF7;
   // UNICODE_TO_GBK[31898] := 16#8980;
   // UNICODE_TO_GBK[31899] := 16#D282;
   // UNICODE_TO_GBK[31900] := 16#8981;
   // UNICODE_TO_GBK[31901] := 16#D2AA;
   // UNICODE_TO_GBK[31902] := 16#8982;
   // UNICODE_TO_GBK[31903] := 16#D283;
   // UNICODE_TO_GBK[31904] := 16#8983;
   // UNICODE_TO_GBK[31905] := 16#F1FB;
   // UNICODE_TO_GBK[31906] := 16#8984;
   // UNICODE_TO_GBK[31907] := 16#D284;
   // UNICODE_TO_GBK[31908] := 16#8985;
   // UNICODE_TO_GBK[31909] := 16#D285;
   // UNICODE_TO_GBK[31910] := 16#8986;
   // UNICODE_TO_GBK[31911] := 16#B8B2;
   // UNICODE_TO_GBK[31912] := 16#8987;
   // UNICODE_TO_GBK[31913] := 16#D286;
   // UNICODE_TO_GBK[31914] := 16#8988;
   // UNICODE_TO_GBK[31915] := 16#D287;
   // UNICODE_TO_GBK[31916] := 16#8989;
   // UNICODE_TO_GBK[31917] := 16#D288;
   // UNICODE_TO_GBK[31918] := 16#898A;
   // UNICODE_TO_GBK[31919] := 16#D289;
   // UNICODE_TO_GBK[31920] := 16#898B;
   // UNICODE_TO_GBK[31921] := 16#D28A;
   // UNICODE_TO_GBK[31922] := 16#898C;
   // UNICODE_TO_GBK[31923] := 16#D28B;
   // UNICODE_TO_GBK[31924] := 16#898D;
   // UNICODE_TO_GBK[31925] := 16#D28C;
   // UNICODE_TO_GBK[31926] := 16#898E;
   // UNICODE_TO_GBK[31927] := 16#D28D;
   // UNICODE_TO_GBK[31928] := 16#898F;
   // UNICODE_TO_GBK[31929] := 16#D28E;
   // UNICODE_TO_GBK[31930] := 16#8990;
   // UNICODE_TO_GBK[31931] := 16#D28F;
   // UNICODE_TO_GBK[31932] := 16#8991;
   // UNICODE_TO_GBK[31933] := 16#D290;
   // UNICODE_TO_GBK[31934] := 16#8992;
   // UNICODE_TO_GBK[31935] := 16#D291;
   // UNICODE_TO_GBK[31936] := 16#8993;
   // UNICODE_TO_GBK[31937] := 16#D292;
   // UNICODE_TO_GBK[31938] := 16#8994;
   // UNICODE_TO_GBK[31939] := 16#D293;
   // UNICODE_TO_GBK[31940] := 16#8995;
   // UNICODE_TO_GBK[31941] := 16#D294;
   // UNICODE_TO_GBK[31942] := 16#8996;
   // UNICODE_TO_GBK[31943] := 16#D295;
   // UNICODE_TO_GBK[31944] := 16#8997;
   // UNICODE_TO_GBK[31945] := 16#D296;
   // UNICODE_TO_GBK[31946] := 16#8998;
   // UNICODE_TO_GBK[31947] := 16#D297;
   // UNICODE_TO_GBK[31948] := 16#8999;
   // UNICODE_TO_GBK[31949] := 16#D298;
   // UNICODE_TO_GBK[31950] := 16#899A;
   // UNICODE_TO_GBK[31951] := 16#D299;
   // UNICODE_TO_GBK[31952] := 16#899B;
   // UNICODE_TO_GBK[31953] := 16#D29A;
   // UNICODE_TO_GBK[31954] := 16#899C;
   // UNICODE_TO_GBK[31955] := 16#D29B;
   // UNICODE_TO_GBK[31956] := 16#899D;
   // UNICODE_TO_GBK[31957] := 16#D29C;
   // UNICODE_TO_GBK[31958] := 16#899E;
   // UNICODE_TO_GBK[31959] := 16#D29D;
   // UNICODE_TO_GBK[31960] := 16#899F;
   // UNICODE_TO_GBK[31961] := 16#D29E;
   // UNICODE_TO_GBK[31962] := 16#89A0;
   // UNICODE_TO_GBK[31963] := 16#D29F;
   // UNICODE_TO_GBK[31964] := 16#89A1;
   // UNICODE_TO_GBK[31965] := 16#D2A0;
   // UNICODE_TO_GBK[31966] := 16#89A2;
   // UNICODE_TO_GBK[31967] := 16#D340;
   // UNICODE_TO_GBK[31968] := 16#89A3;
   // UNICODE_TO_GBK[31969] := 16#D341;
   // UNICODE_TO_GBK[31970] := 16#89A4;
   // UNICODE_TO_GBK[31971] := 16#D342;
   // UNICODE_TO_GBK[31972] := 16#89A5;
   // UNICODE_TO_GBK[31973] := 16#D343;
   // UNICODE_TO_GBK[31974] := 16#89A6;
   // UNICODE_TO_GBK[31975] := 16#D344;
   // UNICODE_TO_GBK[31976] := 16#89A7;
   // UNICODE_TO_GBK[31977] := 16#D345;
   // UNICODE_TO_GBK[31978] := 16#89A8;
   // UNICODE_TO_GBK[31979] := 16#D346;
   // UNICODE_TO_GBK[31980] := 16#89A9;
   // UNICODE_TO_GBK[31981] := 16#D347;
   // UNICODE_TO_GBK[31982] := 16#89AA;
   // UNICODE_TO_GBK[31983] := 16#D348;
   // UNICODE_TO_GBK[31984] := 16#89AB;
   // UNICODE_TO_GBK[31985] := 16#D349;
   // UNICODE_TO_GBK[31986] := 16#89AC;
   // UNICODE_TO_GBK[31987] := 16#D34A;
   // UNICODE_TO_GBK[31988] := 16#89AD;
   // UNICODE_TO_GBK[31989] := 16#D34B;
   // UNICODE_TO_GBK[31990] := 16#89AE;
   // UNICODE_TO_GBK[31991] := 16#D34C;
   // UNICODE_TO_GBK[31992] := 16#89AF;
   // UNICODE_TO_GBK[31993] := 16#D34D;
   // UNICODE_TO_GBK[31994] := 16#89B0;
   // UNICODE_TO_GBK[31995] := 16#D34E;
   // UNICODE_TO_GBK[31996] := 16#89B1;
   // UNICODE_TO_GBK[31997] := 16#D34F;
   // UNICODE_TO_GBK[31998] := 16#89B2;
   // UNICODE_TO_GBK[31999] := 16#D350;
   // UNICODE_TO_GBK[32000] := 16#89B3;
   // UNICODE_TO_GBK[32001] := 16#D351;
   // UNICODE_TO_GBK[32002] := 16#89B4;
   // UNICODE_TO_GBK[32003] := 16#D352;
   // UNICODE_TO_GBK[32004] := 16#89B5;
   // UNICODE_TO_GBK[32005] := 16#D353;
   // UNICODE_TO_GBK[32006] := 16#89B6;
   // UNICODE_TO_GBK[32007] := 16#D354;
   // UNICODE_TO_GBK[32008] := 16#89B7;
   // UNICODE_TO_GBK[32009] := 16#D355;
   // UNICODE_TO_GBK[32010] := 16#89B8;
   // UNICODE_TO_GBK[32011] := 16#D356;
   // UNICODE_TO_GBK[32012] := 16#89B9;
   // UNICODE_TO_GBK[32013] := 16#D357;
   // UNICODE_TO_GBK[32014] := 16#89BA;
   // UNICODE_TO_GBK[32015] := 16#D358;
   // UNICODE_TO_GBK[32016] := 16#89BB;
   // UNICODE_TO_GBK[32017] := 16#D359;
   // UNICODE_TO_GBK[32018] := 16#89BC;
   // UNICODE_TO_GBK[32019] := 16#D35A;
   // UNICODE_TO_GBK[32020] := 16#89BD;
   // UNICODE_TO_GBK[32021] := 16#D35B;
   // UNICODE_TO_GBK[32022] := 16#89BE;
   // UNICODE_TO_GBK[32023] := 16#D35C;
   // UNICODE_TO_GBK[32024] := 16#89BF;
   // UNICODE_TO_GBK[32025] := 16#D35D;
   // UNICODE_TO_GBK[32026] := 16#89C0;
   // UNICODE_TO_GBK[32027] := 16#D35E;
   // UNICODE_TO_GBK[32028] := 16#89C1;
   // UNICODE_TO_GBK[32029] := 16#BCFB;
   // UNICODE_TO_GBK[32030] := 16#89C2;
   // UNICODE_TO_GBK[32031] := 16#B9DB;
   // UNICODE_TO_GBK[32032] := 16#89C3;
   // UNICODE_TO_GBK[32033] := 16#D35F;
   // UNICODE_TO_GBK[32034] := 16#89C4;
   // UNICODE_TO_GBK[32035] := 16#B9E6;
   // UNICODE_TO_GBK[32036] := 16#89C5;
   // UNICODE_TO_GBK[32037] := 16#C3D9;
   // UNICODE_TO_GBK[32038] := 16#89C6;
   // UNICODE_TO_GBK[32039] := 16#CAD3;
   // UNICODE_TO_GBK[32040] := 16#89C7;
   // UNICODE_TO_GBK[32041] := 16#EAE8;
   // UNICODE_TO_GBK[32042] := 16#89C8;
   // UNICODE_TO_GBK[32043] := 16#C0C0;
   // UNICODE_TO_GBK[32044] := 16#89C9;
   // UNICODE_TO_GBK[32045] := 16#BEF5;
   // UNICODE_TO_GBK[32046] := 16#89CA;
   // UNICODE_TO_GBK[32047] := 16#EAE9;
   // UNICODE_TO_GBK[32048] := 16#89CB;
   // UNICODE_TO_GBK[32049] := 16#EAEA;
   // UNICODE_TO_GBK[32050] := 16#89CC;
   // UNICODE_TO_GBK[32051] := 16#EAEB;
   // UNICODE_TO_GBK[32052] := 16#89CD;
   // UNICODE_TO_GBK[32053] := 16#D360;
   // UNICODE_TO_GBK[32054] := 16#89CE;
   // UNICODE_TO_GBK[32055] := 16#EAEC;
   // UNICODE_TO_GBK[32056] := 16#89CF;
   // UNICODE_TO_GBK[32057] := 16#EAED;
   // UNICODE_TO_GBK[32058] := 16#89D0;
   // UNICODE_TO_GBK[32059] := 16#EAEE;
   // UNICODE_TO_GBK[32060] := 16#89D1;
   // UNICODE_TO_GBK[32061] := 16#EAEF;
   // UNICODE_TO_GBK[32062] := 16#89D2;
   // UNICODE_TO_GBK[32063] := 16#BDC7;
   // UNICODE_TO_GBK[32064] := 16#89D3;
   // UNICODE_TO_GBK[32065] := 16#D361;
   // UNICODE_TO_GBK[32066] := 16#89D4;
   // UNICODE_TO_GBK[32067] := 16#D362;
   // UNICODE_TO_GBK[32068] := 16#89D5;
   // UNICODE_TO_GBK[32069] := 16#D363;
   // UNICODE_TO_GBK[32070] := 16#89D6;
   // UNICODE_TO_GBK[32071] := 16#F5FB;
   // UNICODE_TO_GBK[32072] := 16#89D7;
   // UNICODE_TO_GBK[32073] := 16#D364;
   // UNICODE_TO_GBK[32074] := 16#89D8;
   // UNICODE_TO_GBK[32075] := 16#D365;
   // UNICODE_TO_GBK[32076] := 16#89D9;
   // UNICODE_TO_GBK[32077] := 16#D366;
   // UNICODE_TO_GBK[32078] := 16#89DA;
   // UNICODE_TO_GBK[32079] := 16#F5FD;
   // UNICODE_TO_GBK[32080] := 16#89DB;
   // UNICODE_TO_GBK[32081] := 16#D367;
   // UNICODE_TO_GBK[32082] := 16#89DC;
   // UNICODE_TO_GBK[32083] := 16#F5FE;
   // UNICODE_TO_GBK[32084] := 16#89DD;
   // UNICODE_TO_GBK[32085] := 16#D368;
   // UNICODE_TO_GBK[32086] := 16#89DE;
   // UNICODE_TO_GBK[32087] := 16#F5FC;
   // UNICODE_TO_GBK[32088] := 16#89DF;
   // UNICODE_TO_GBK[32089] := 16#D369;
   // UNICODE_TO_GBK[32090] := 16#89E0;
   // UNICODE_TO_GBK[32091] := 16#D36A;
   // UNICODE_TO_GBK[32092] := 16#89E1;
   // UNICODE_TO_GBK[32093] := 16#D36B;
   // UNICODE_TO_GBK[32094] := 16#89E2;
   // UNICODE_TO_GBK[32095] := 16#D36C;
   // UNICODE_TO_GBK[32096] := 16#89E3;
   // UNICODE_TO_GBK[32097] := 16#BDE2;
   // UNICODE_TO_GBK[32098] := 16#89E4;
   // UNICODE_TO_GBK[32099] := 16#D36D;
   // UNICODE_TO_GBK[32100] := 16#89E5;
   // UNICODE_TO_GBK[32101] := 16#F6A1;
   // UNICODE_TO_GBK[32102] := 16#89E6;
   // UNICODE_TO_GBK[32103] := 16#B4A5;
   // UNICODE_TO_GBK[32104] := 16#89E7;
   // UNICODE_TO_GBK[32105] := 16#D36E;
   // UNICODE_TO_GBK[32106] := 16#89E8;
   // UNICODE_TO_GBK[32107] := 16#D36F;
   // UNICODE_TO_GBK[32108] := 16#89E9;
   // UNICODE_TO_GBK[32109] := 16#D370;
   // UNICODE_TO_GBK[32110] := 16#89EA;
   // UNICODE_TO_GBK[32111] := 16#D371;
   // UNICODE_TO_GBK[32112] := 16#89EB;
   // UNICODE_TO_GBK[32113] := 16#F6A2;
   // UNICODE_TO_GBK[32114] := 16#89EC;
   // UNICODE_TO_GBK[32115] := 16#D372;
   // UNICODE_TO_GBK[32116] := 16#89ED;
   // UNICODE_TO_GBK[32117] := 16#D373;
   // UNICODE_TO_GBK[32118] := 16#89EE;
   // UNICODE_TO_GBK[32119] := 16#D374;
   // UNICODE_TO_GBK[32120] := 16#89EF;
   // UNICODE_TO_GBK[32121] := 16#F6A3;
   // UNICODE_TO_GBK[32122] := 16#89F0;
   // UNICODE_TO_GBK[32123] := 16#D375;
   // UNICODE_TO_GBK[32124] := 16#89F1;
   // UNICODE_TO_GBK[32125] := 16#D376;
   // UNICODE_TO_GBK[32126] := 16#89F2;
   // UNICODE_TO_GBK[32127] := 16#D377;
   // UNICODE_TO_GBK[32128] := 16#89F3;
   // UNICODE_TO_GBK[32129] := 16#ECB2;
   // UNICODE_TO_GBK[32130] := 16#89F4;
   // UNICODE_TO_GBK[32131] := 16#D378;
   // UNICODE_TO_GBK[32132] := 16#89F5;
   // UNICODE_TO_GBK[32133] := 16#D379;
   // UNICODE_TO_GBK[32134] := 16#89F6;
   // UNICODE_TO_GBK[32135] := 16#D37A;
   // UNICODE_TO_GBK[32136] := 16#89F7;
   // UNICODE_TO_GBK[32137] := 16#D37B;
   // UNICODE_TO_GBK[32138] := 16#89F8;
   // UNICODE_TO_GBK[32139] := 16#D37C;
   // UNICODE_TO_GBK[32140] := 16#89F9;
   // UNICODE_TO_GBK[32141] := 16#D37D;
   // UNICODE_TO_GBK[32142] := 16#89FA;
   // UNICODE_TO_GBK[32143] := 16#D37E;
   // UNICODE_TO_GBK[32144] := 16#89FB;
   // UNICODE_TO_GBK[32145] := 16#D380;
   // UNICODE_TO_GBK[32146] := 16#89FC;
   // UNICODE_TO_GBK[32147] := 16#D381;
   // UNICODE_TO_GBK[32148] := 16#89FD;
   // UNICODE_TO_GBK[32149] := 16#D382;
   // UNICODE_TO_GBK[32150] := 16#89FE;
   // UNICODE_TO_GBK[32151] := 16#D383;
   // UNICODE_TO_GBK[32152] := 16#89FF;
   // UNICODE_TO_GBK[32153] := 16#D384;
   // UNICODE_TO_GBK[32154] := 16#8A00;
   // UNICODE_TO_GBK[32155] := 16#D1D4;
   // UNICODE_TO_GBK[32156] := 16#8A01;
   // UNICODE_TO_GBK[32157] := 16#D385;
   // UNICODE_TO_GBK[32158] := 16#8A02;
   // UNICODE_TO_GBK[32159] := 16#D386;
   // UNICODE_TO_GBK[32160] := 16#8A03;
   // UNICODE_TO_GBK[32161] := 16#D387;
   // UNICODE_TO_GBK[32162] := 16#8A04;
   // UNICODE_TO_GBK[32163] := 16#D388;
   // UNICODE_TO_GBK[32164] := 16#8A05;
   // UNICODE_TO_GBK[32165] := 16#D389;
   // UNICODE_TO_GBK[32166] := 16#8A06;
   // UNICODE_TO_GBK[32167] := 16#D38A;
   // UNICODE_TO_GBK[32168] := 16#8A07;
   // UNICODE_TO_GBK[32169] := 16#D9EA;
   // UNICODE_TO_GBK[32170] := 16#8A08;
   // UNICODE_TO_GBK[32171] := 16#D38B;
   // UNICODE_TO_GBK[32172] := 16#8A09;
   // UNICODE_TO_GBK[32173] := 16#D38C;
   // UNICODE_TO_GBK[32174] := 16#8A0A;
   // UNICODE_TO_GBK[32175] := 16#D38D;
   // UNICODE_TO_GBK[32176] := 16#8A0B;
   // UNICODE_TO_GBK[32177] := 16#D38E;
   // UNICODE_TO_GBK[32178] := 16#8A0C;
   // UNICODE_TO_GBK[32179] := 16#D38F;
   // UNICODE_TO_GBK[32180] := 16#8A0D;
   // UNICODE_TO_GBK[32181] := 16#D390;
   // UNICODE_TO_GBK[32182] := 16#8A0E;
   // UNICODE_TO_GBK[32183] := 16#D391;
   // UNICODE_TO_GBK[32184] := 16#8A0F;
   // UNICODE_TO_GBK[32185] := 16#D392;
   // UNICODE_TO_GBK[32186] := 16#8A10;
   // UNICODE_TO_GBK[32187] := 16#D393;
   // UNICODE_TO_GBK[32188] := 16#8A11;
   // UNICODE_TO_GBK[32189] := 16#D394;
   // UNICODE_TO_GBK[32190] := 16#8A12;
   // UNICODE_TO_GBK[32191] := 16#D395;
   // UNICODE_TO_GBK[32192] := 16#8A13;
   // UNICODE_TO_GBK[32193] := 16#D396;
   // UNICODE_TO_GBK[32194] := 16#8A14;
   // UNICODE_TO_GBK[32195] := 16#D397;
   // UNICODE_TO_GBK[32196] := 16#8A15;
   // UNICODE_TO_GBK[32197] := 16#D398;
   // UNICODE_TO_GBK[32198] := 16#8A16;
   // UNICODE_TO_GBK[32199] := 16#D399;
   // UNICODE_TO_GBK[32200] := 16#8A17;
   // UNICODE_TO_GBK[32201] := 16#D39A;
   // UNICODE_TO_GBK[32202] := 16#8A18;
   // UNICODE_TO_GBK[32203] := 16#D39B;
   // UNICODE_TO_GBK[32204] := 16#8A19;
   // UNICODE_TO_GBK[32205] := 16#D39C;
   // UNICODE_TO_GBK[32206] := 16#8A1A;
   // UNICODE_TO_GBK[32207] := 16#D39D;
   // UNICODE_TO_GBK[32208] := 16#8A1B;
   // UNICODE_TO_GBK[32209] := 16#D39E;
   // UNICODE_TO_GBK[32210] := 16#8A1C;
   // UNICODE_TO_GBK[32211] := 16#D39F;
   // UNICODE_TO_GBK[32212] := 16#8A1D;
   // UNICODE_TO_GBK[32213] := 16#D3A0;
   // UNICODE_TO_GBK[32214] := 16#8A1E;
   // UNICODE_TO_GBK[32215] := 16#D440;
   // UNICODE_TO_GBK[32216] := 16#8A1F;
   // UNICODE_TO_GBK[32217] := 16#D441;
   // UNICODE_TO_GBK[32218] := 16#8A20;
   // UNICODE_TO_GBK[32219] := 16#D442;
   // UNICODE_TO_GBK[32220] := 16#8A21;
   // UNICODE_TO_GBK[32221] := 16#D443;
   // UNICODE_TO_GBK[32222] := 16#8A22;
   // UNICODE_TO_GBK[32223] := 16#D444;
   // UNICODE_TO_GBK[32224] := 16#8A23;
   // UNICODE_TO_GBK[32225] := 16#D445;
   // UNICODE_TO_GBK[32226] := 16#8A24;
   // UNICODE_TO_GBK[32227] := 16#D446;
   // UNICODE_TO_GBK[32228] := 16#8A25;
   // UNICODE_TO_GBK[32229] := 16#D447;
   // UNICODE_TO_GBK[32230] := 16#8A26;
   // UNICODE_TO_GBK[32231] := 16#D448;
   // UNICODE_TO_GBK[32232] := 16#8A27;
   // UNICODE_TO_GBK[32233] := 16#D449;
   // UNICODE_TO_GBK[32234] := 16#8A28;
   // UNICODE_TO_GBK[32235] := 16#D44A;
   // UNICODE_TO_GBK[32236] := 16#8A29;
   // UNICODE_TO_GBK[32237] := 16#D44B;
   // UNICODE_TO_GBK[32238] := 16#8A2A;
   // UNICODE_TO_GBK[32239] := 16#D44C;
   // UNICODE_TO_GBK[32240] := 16#8A2B;
   // UNICODE_TO_GBK[32241] := 16#D44D;
   // UNICODE_TO_GBK[32242] := 16#8A2C;
   // UNICODE_TO_GBK[32243] := 16#D44E;
   // UNICODE_TO_GBK[32244] := 16#8A2D;
   // UNICODE_TO_GBK[32245] := 16#D44F;
   // UNICODE_TO_GBK[32246] := 16#8A2E;
   // UNICODE_TO_GBK[32247] := 16#D450;
   // UNICODE_TO_GBK[32248] := 16#8A2F;
   // UNICODE_TO_GBK[32249] := 16#D451;
   // UNICODE_TO_GBK[32250] := 16#8A30;
   // UNICODE_TO_GBK[32251] := 16#D452;
   // UNICODE_TO_GBK[32252] := 16#8A31;
   // UNICODE_TO_GBK[32253] := 16#D453;
   // UNICODE_TO_GBK[32254] := 16#8A32;
   // UNICODE_TO_GBK[32255] := 16#D454;
   // UNICODE_TO_GBK[32256] := 16#8A33;
   // UNICODE_TO_GBK[32257] := 16#D455;
   // UNICODE_TO_GBK[32258] := 16#8A34;
   // UNICODE_TO_GBK[32259] := 16#D456;
   // UNICODE_TO_GBK[32260] := 16#8A35;
   // UNICODE_TO_GBK[32261] := 16#D457;
   // UNICODE_TO_GBK[32262] := 16#8A36;
   // UNICODE_TO_GBK[32263] := 16#D458;
   // UNICODE_TO_GBK[32264] := 16#8A37;
   // UNICODE_TO_GBK[32265] := 16#D459;
   // UNICODE_TO_GBK[32266] := 16#8A38;
   // UNICODE_TO_GBK[32267] := 16#D45A;
   // UNICODE_TO_GBK[32268] := 16#8A39;
   // UNICODE_TO_GBK[32269] := 16#D45B;
   // UNICODE_TO_GBK[32270] := 16#8A3A;
   // UNICODE_TO_GBK[32271] := 16#D45C;
   // UNICODE_TO_GBK[32272] := 16#8A3B;
   // UNICODE_TO_GBK[32273] := 16#D45D;
   // UNICODE_TO_GBK[32274] := 16#8A3C;
   // UNICODE_TO_GBK[32275] := 16#D45E;
   // UNICODE_TO_GBK[32276] := 16#8A3D;
   // UNICODE_TO_GBK[32277] := 16#D45F;
   // UNICODE_TO_GBK[32278] := 16#8A3E;
   // UNICODE_TO_GBK[32279] := 16#F6A4;
   // UNICODE_TO_GBK[32280] := 16#8A3F;
   // UNICODE_TO_GBK[32281] := 16#D460;
   // UNICODE_TO_GBK[32282] := 16#8A40;
   // UNICODE_TO_GBK[32283] := 16#D461;
   // UNICODE_TO_GBK[32284] := 16#8A41;
   // UNICODE_TO_GBK[32285] := 16#D462;
   // UNICODE_TO_GBK[32286] := 16#8A42;
   // UNICODE_TO_GBK[32287] := 16#D463;
   // UNICODE_TO_GBK[32288] := 16#8A43;
   // UNICODE_TO_GBK[32289] := 16#D464;
   // UNICODE_TO_GBK[32290] := 16#8A44;
   // UNICODE_TO_GBK[32291] := 16#D465;
   // UNICODE_TO_GBK[32292] := 16#8A45;
   // UNICODE_TO_GBK[32293] := 16#D466;
   // UNICODE_TO_GBK[32294] := 16#8A46;
   // UNICODE_TO_GBK[32295] := 16#D467;
   // UNICODE_TO_GBK[32296] := 16#8A47;
   // UNICODE_TO_GBK[32297] := 16#D468;
   // UNICODE_TO_GBK[32298] := 16#8A48;
   // UNICODE_TO_GBK[32299] := 16#EEBA;
   // UNICODE_TO_GBK[32300] := 16#8A49;
   // UNICODE_TO_GBK[32301] := 16#D469;
   // UNICODE_TO_GBK[32302] := 16#8A4A;
   // UNICODE_TO_GBK[32303] := 16#D46A;
   // UNICODE_TO_GBK[32304] := 16#8A4B;
   // UNICODE_TO_GBK[32305] := 16#D46B;
   // UNICODE_TO_GBK[32306] := 16#8A4C;
   // UNICODE_TO_GBK[32307] := 16#D46C;
   // UNICODE_TO_GBK[32308] := 16#8A4D;
   // UNICODE_TO_GBK[32309] := 16#D46D;
   // UNICODE_TO_GBK[32310] := 16#8A4E;
   // UNICODE_TO_GBK[32311] := 16#D46E;
   // UNICODE_TO_GBK[32312] := 16#8A4F;
   // UNICODE_TO_GBK[32313] := 16#D46F;
   // UNICODE_TO_GBK[32314] := 16#8A50;
   // UNICODE_TO_GBK[32315] := 16#D470;
   // UNICODE_TO_GBK[32316] := 16#8A51;
   // UNICODE_TO_GBK[32317] := 16#D471;
   // UNICODE_TO_GBK[32318] := 16#8A52;
   // UNICODE_TO_GBK[32319] := 16#D472;
   // UNICODE_TO_GBK[32320] := 16#8A53;
   // UNICODE_TO_GBK[32321] := 16#D473;
   // UNICODE_TO_GBK[32322] := 16#8A54;
   // UNICODE_TO_GBK[32323] := 16#D474;
   // UNICODE_TO_GBK[32324] := 16#8A55;
   // UNICODE_TO_GBK[32325] := 16#D475;
